LIN {X 0.222,Y -452.244,Z 357.481,A 0.000,B 0.000,C 90.000,E1 266.502} C_DIS
LIN {X -0.089,Y -444.723,Z 357.479,A 0.000,B 0.000,C 90.000,E1 266.274} C_DIS
LIN {X 0.117,Y -436.649,Z 357.478,A 0.000,B 0.000,C 90.000,E1 266.045} C_DIS
LIN {X -0.080,Y -427.748,Z 357.477,A 0.000,B 0.000,C 90.000,E1 265.927} C_DIS
LIN {X 0.197,Y -418.115,Z 357.477,A 0.000,B 0.000,C 90.000,E1 265.812} C_DIS
LIN {X 0.128,Y -415.170,Z 357.477,A 0.000,B 0.000,C 90.000,E1 265.812} C_DIS
LIN {X 0.027,Y -180.914,Z 357.477,A 0.000,B 0.000,C 90.000,E1 265.812} C_DIS
LIN {X -0.032,Y -180.848,Z 357.472,A 0.000,B 0.000,C 90.000,E1 264.951} C_DIS
LIN {X 0.050,Y -178.957,Z 357.444,A 0.000,B 0.000,C 90.000,E1 259.859} C_DIS
LIN {X -0.057,Y -177.360,Z 357.430,A 0.000,B 0.000,C 90.000,E1 257.353} C_DIS
LIN {X 0.039,Y -175.531,Z 357.411,A 0.000,B 0.000,C 90.000,E1 253.921} C_DIS
LIN {X 0.040,Y -172.266,Z 357.387,A 0.000,B 0.000,C 90.000,E1 249.645} C_DIS
LIN {X 0.079,Y -171.746,Z 357.382,A 0.000,B 0.000,C 90.000,E1 248.773} C_DIS
LIN {X -0.063,Y -167.343,Z 357.353,A 0.000,B 0.000,C 90.000,E1 243.640} C_DIS
LIN {X 0.018,Y -166.730,Z 357.349,A 0.000,B 0.000,C 90.000,E1 242.743} C_DIS
LIN {X -0.069,Y -162.709,Z 357.324,A 0.000,B 0.000,C 90.000,E1 238.408} C_DIS
LIN {X -0.007,Y -161.400,Z 357.315,A 0.000,B 0.000,C 90.000,E1 236.628} C_DIS
LIN {X 0.035,Y -157.393,Z 357.290,A 0.000,B 0.000,C 90.000,E1 232.190} C_DIS
LIN {X -0.032,Y -155.390,Z 357.275,A 0.000,B 0.000,C 90.000,E1 229.542} C_DIS
LIN {X 0.007,Y -151.724,Z 357.250,A 0.000,B 0.000,C 90.000,E1 225.040} C_DIS
LIN {X 0.023,Y -149.918,Z 357.235,A 0.000,B 0.000,C 90.000,E1 222.324} C_DIS
LIN {X -0.059,Y -146.773,Z 357.210,A 0.000,B 0.000,C 90.000,E1 217.810} C_DIS
LIN {X 0.045,Y -145.342,Z 357.195,A 0.000,B 0.000,C 90.000,E1 215.025} C_DIS
LIN {X -0.040,Y -142.418,Z 357.164,A 0.000,B 0.000,C 90.000,E1 209.539} C_DIS
LIN {X 0.009,Y -141.404,Z 357.149,A 0.000,B 0.000,C 90.000,E1 206.744} C_DIS
LIN {X -0.003,Y -139.356,Z 357.112,A 0.000,B 0.000,C 90.000,E1 200.248} C_DIS
LIN {X -0.015,Y -138.798,Z 357.097,A 0.000,B 0.000,C 90.000,E1 197.457} C_DIS
LIN {X 0.039,Y -138.348,Z 357.055,A 0.000,B 0.000,C 90.000,E1 189.962} C_DIS
LIN {X 0.057,Y -139.371,Z 357.009,A 0.000,B 0.000,C 90.000,E1 181.547} C_DIS
LIN {X -0.029,Y -141.260,Z 356.973,A 0.000,B 0.000,C 90.000,E1 175.065} C_DIS
LIN {X -0.071,Y -142.628,Z 356.957,A 0.000,B 0.000,C 90.000,E1 172.299} C_DIS
LIN {X 0.022,Y -144.952,Z 356.931,A 0.000,B 0.000,C 90.000,E1 167.645} C_DIS
LIN {X 0.013,Y -147.581,Z 356.911,A 0.000,B 0.000,C 90.000,E1 163.976} C_DIS
LIN {X 0.044,Y -150.192,Z 356.891,A 0.000,B 0.000,C 90.000,E1 160.315} C_DIS
LIN {X -0.030,Y -153.574,Z 356.871,A 0.000,B 0.000,C 90.000,E1 156.719} C_DIS
LIN {X -0.039,Y -156.991,Z 356.851,A 0.000,B 0.000,C 90.000,E1 153.127} C_DIS
LIN {X 0.034,Y -161.105,Z 356.831,A 0.000,B 0.000,C 90.000,E1 149.537} C_DIS
LIN {X -0.021,Y -163.208,Z 356.821,A 0.000,B 0.000,C 90.000,E1 147.788} C_DIS
LIN {X -0.016,Y -167.635,Z 356.802,A 0.000,B 0.000,C 90.000,E1 144.276} C_DIS
LIN {X -0.001,Y -171.461,Z 356.787,A 0.000,B 0.000,C 90.000,E1 141.662} C_DIS
LIN {X -0.071,Y -176.386,Z 356.768,A 0.000,B 0.000,C 90.000,E1 138.243} C_DIS
LIN {X 0.051,Y -180.680,Z 356.754,A 0.000,B 0.000,C 90.000,E1 135.648} C_DIS
LIN {X 0.033,Y -186.082,Z 356.735,A 0.000,B 0.000,C 90.000,E1 132.285} C_DIS
LIN {X -0.030,Y -190.719,Z 356.721,A 0.000,B 0.000,C 90.000,E1 129.806} C_DIS
LIN {X 0.001,Y -196.472,Z 356.703,A 0.000,B 0.000,C 90.000,E1 126.503} C_DIS
LIN {X 0.023,Y -199.896,Z 356.693,A 0.000,B 0.000,C 90.000,E1 124.771} C_DIS
LIN {X -0.019,Y -300.209,Z 356.693,A 0.000,B 0.000,C 90.000,E1 124.771} C_DIS
LIN {X -0.007,Y -301.841,Z 356.693,A 0.000,B 0.000,C 90.000,E1 124.739} C_DIS
LIN {X 0.022,Y -305.622,Z 356.692,A 0.000,B 0.000,C 90.000,E1 124.565} C_DIS
LIN {X -0.029,Y -307.838,Z 356.691,A 0.000,B 0.000,C 90.000,E1 124.405} C_DIS
LIN {X -0.050,Y -310.913,Z 356.689,A 0.000,B 0.000,C 90.000,E1 124.072} C_DIS
LIN {X -0.137,Y -312.908,Z 356.688,A 0.000,B 0.000,C 90.000,E1 123.785} C_DIS
LIN {X 0.036,Y -314.472,Z 356.686,A 0.000,B 0.000,C 90.000,E1 123.452} C_DIS
LIN {X -0.111,Y -316.907,Z 356.682,A 0.000,B 0.000,C 90.000,E1 122.832} C_DIS
LIN {X 0.081,Y -327.434,Z 356.666,A 0.000,B 0.000,C 90.000,E1 119.922} C_DIS
LIN {X -0.084,Y -339.335,Z 356.651,A 0.000,B 0.000,C 90.000,E1 117.129} C_DIS
LIN {X 0.101,Y -352.712,Z 356.635,A 0.000,B 0.000,C 90.000,E1 114.335} C_DIS
LIN {X -0.020,Y -365.944,Z 356.622,A 0.000,B 0.000,C 90.000,E1 111.950} C_DIS
LIN {X 0.123,Y -380.539,Z 356.609,A 0.000,B 0.000,C 90.000,E1 109.577} C_DIS
LIN {X 0.160,Y -396.602,Z 356.596,A 0.000,B 0.000,C 90.000,E1 107.275} C_DIS
LIN {X -0.034,Y -414.254,Z 356.584,A 0.000,B 0.000,C 90.000,E1 105.064} C_DIS
LIN {X 0.018,Y -433.580,Z 356.572,A 0.000,B 0.000,C 90.000,E1 102.883} C_DIS
LIN {X 0.187,Y -453.825,Z 356.560,A 0.000,B 0.000,C 90.000,E1 100.838} C_DIS
LIN {X -0.188,Y -474.606,Z 356.550,A 0.000,B 0.000,C 90.000,E1 99.029} C_DIS
LIN {X -0.195,Y -492.986,Z 356.542,A 0.000,B 0.000,C 90.000,E1 97.530} C_DIS
LIN {X 0.033,Y -496.458,Z 356.539,A 0.000,B 0.000,C 90.000,E1 97.068} C_DIS
LIN {X -0.061,Y -497.755,Z 356.538,A 0.000,B 0.000,C 90.000,E1 96.834} C_DIS
LIN {X -0.215,Y -498.705,Z 356.537,A 0.000,B 0.000,C 90.000,E1 96.606} C_DIS
LIN {X 0.058,Y -499.740,Z 356.534,A 0.000,B 0.000,C 90.000,E1 96.087} C_DIS
LIN {X -0.161,Y -499.759,Z 356.531,A 0.000,B 0.000,C 90.000,E1 95.625} C_DIS
LIN {X 0.121,Y -498.765,Z 356.528,A 0.000,B 0.000,C 90.000,E1 95.106} C_DIS
LIN {X -0.008,Y -497.842,Z 356.527,A 0.000,B 0.000,C 90.000,E1 94.878} C_DIS
LIN {X -0.095,Y -496.578,Z 356.526,A 0.000,B 0.000,C 90.000,E1 94.645} C_DIS
LIN {X 0.031,Y -491.350,Z 356.522,A 0.000,B 0.000,C 90.000,E1 93.898} C_DIS
LIN {X -0.040,Y -483.657,Z 356.516,A 0.000,B 0.000,C 90.000,E1 92.922} C_DIS
LIN {X 0.090,Y -463.710,Z 356.502,A 0.000,B 0.000,C 90.000,E1 90.401} C_DIS
LIN {X 0.125,Y -445.143,Z 356.488,A 0.000,B 0.000,C 90.000,E1 87.822} C_DIS
LIN {X -0.162,Y -426.612,Z 356.472,A 0.000,B 0.000,C 90.000,E1 84.951} C_DIS
LIN {X 0.108,Y -406.776,Z 356.452,A 0.000,B 0.000,C 90.000,E1 81.376} C_DIS
LIN {X -0.002,Y -395.068,Z 356.440,A 0.000,B 0.000,C 90.000,E1 79.162} C_DIS
LIN {X 0.039,Y -384.866,Z 356.429,A 0.000,B 0.000,C 90.000,E1 77.173} C_DIS
LIN {X 0.046,Y -373.237,Z 356.416,A 0.000,B 0.000,C 90.000,E1 74.866} C_DIS
LIN {X -0.124,Y -361.668,Z 356.403,A 0.000,B 0.000,C 90.000,E1 72.543} C_DIS
LIN {X 0.054,Y -351.512,Z 356.391,A 0.000,B 0.000,C 90.000,E1 70.423} C_DIS
LIN {X 0.148,Y -337.364,Z 356.374,A 0.000,B 0.000,C 90.000,E1 67.358} C_DIS
LIN {X -0.164,Y -326.775,Z 356.361,A 0.000,B 0.000,C 90.000,E1 64.921} C_DIS
LIN {X 0.063,Y -315.883,Z 356.345,A 0.000,B 0.000,C 90.000,E1 62.025} C_DIS
LIN {X 0.088,Y -303.361,Z 356.325,A 0.000,B 0.000,C 90.000,E1 58.456} C_DIS
LIN {X -0.062,Y -291.846,Z 356.305,A 0.000,B 0.000,C 90.000,E1 54.848} C_DIS
LIN {X 0.046,Y -282.258,Z 356.286,A 0.000,B 0.000,C 90.000,E1 51.457} C_DIS
LIN {X -0.006,Y -274.758,Z 356.271,A 0.000,B 0.000,C 90.000,E1 48.728} C_DIS
LIN {X -0.073,Y -269.054,Z 356.259,A 0.000,B 0.000,C 90.000,E1 46.662} C_DIS
LIN {X -0.126,Y -261.490,Z 356.244,A 0.000,B 0.000,C 90.000,E1 43.866} C_DIS
LIN {X 0.125,Y -255.793,Z 356.232,A 0.000,B 0.000,C 90.000,E1 41.676} C_DIS
LIN {X -0.072,Y -250.024,Z 356.220,A 0.000,B 0.000,C 90.000,E1 39.564} C_DIS
LIN {X 0.010,Y -244.096,Z 356.208,A 0.000,B 0.000,C 90.000,E1 37.363} C_DIS
LIN {X 0.041,Y -236.316,Z 356.191,A 0.000,B 0.000,C 90.000,E1 34.405} C_DIS
LIN {X 0.010,Y -228.739,Z 356.175,A 0.000,B 0.000,C 90.000,E1 31.416} C_DIS
LIN {X 0.063,Y -221.644,Z 356.158,A 0.000,B 0.000,C 90.000,E1 28.359} C_DIS
LIN {X -0.026,Y -213.645,Z 356.136,A 0.000,B 0.000,C 90.000,E1 24.515} C_DIS
LIN {X 0.048,Y -207.922,Z 356.119,A 0.000,B 0.000,C 90.000,E1 21.354} C_DIS
LIN {X 0.025,Y -202.976,Z 356.101,A 0.000,B 0.000,C 90.000,E1 18.181} C_DIS
LIN {X 0.076,Y -198.614,Z 356.083,A 0.000,B 0.000,C 90.000,E1 14.954} C_DIS
LIN {X 0.078,Y -194.085,Z 356.061,A 0.000,B 0.000,C 90.000,E1 10.894} C_DIS
LIN {X -0.046,Y -190.735,Z 356.038,A 0.000,B 0.000,C 90.000,E1 6.834} C_DIS
LIN {X 0.022,Y -188.091,Z 356.006,A 0.000,B 0.000,C 90.000,E1 1.031} C_DIS
LIN {X 0.029,Y -189.258,Z 355.942,A 0.000,B 0.000,C 90.000,E1 349.567} C_DIS
LIN {X -0.030,Y -192.110,Z 355.915,A 0.000,B 0.000,C 90.000,E1 344.629} C_DIS
LIN {X 0.073,Y -195.713,Z 355.892,A 0.000,B 0.000,C 90.000,E1 340.496} C_DIS
LIN {X 0.058,Y -200.400,Z 355.869,A 0.000,B 0.000,C 90.000,E1 336.433} C_DIS
LIN {X 0.058,Y -206.128,Z 355.847,A 0.000,B 0.000,C 90.000,E1 332.410} C_DIS
LIN {X -0.011,Y -212.845,Z 355.825,A 0.000,B 0.000,C 90.000,E1 328.456} C_DIS
LIN {X -0.091,Y -220.250,Z 355.803,A 0.000,B 0.000,C 90.000,E1 324.562} C_DIS
LIN {X 0.033,Y -228.477,Z 355.782,A 0.000,B 0.000,C 90.000,E1 320.678} C_DIS
LIN {X 0.079,Y -235.880,Z 355.765,A 0.000,B 0.000,C 90.000,E1 317.634} C_DIS
LIN {X 0.126,Y -245.235,Z 355.746,A 0.000,B 0.000,C 90.000,E1 314.271} C_DIS
LIN {X 0.123,Y -255.868,Z 355.728,A 0.000,B 0.000,C 90.000,E1 310.987} C_DIS
LIN {X -0.051,Y -267.304,Z 355.710,A 0.000,B 0.000,C 90.000,E1 307.810} C_DIS
LIN {X -0.024,Y -279.759,Z 355.693,A 0.000,B 0.000,C 90.000,E1 304.659} C_DIS
LIN {X -0.037,Y -293.589,Z 355.675,A 0.000,B 0.000,C 90.000,E1 301.592} C_DIS
LIN {X -0.071,Y -310.841,Z 355.657,A 0.000,B 0.000,C 90.000,E1 298.281} C_DIS
LIN {X -0.109,Y -320.424,Z 355.648,A 0.000,B 0.000,C 90.000,E1 296.668} C_DIS
LIN {X -0.141,Y -341.506,Z 355.630,A 0.000,B 0.000,C 90.000,E1 293.515} C_DIS
LIN {X -0.076,Y -354.944,Z 355.620,A 0.000,B 0.000,C 90.000,E1 291.663} C_DIS
LIN {X -0.135,Y -371.202,Z 355.609,A 0.000,B 0.000,C 90.000,E1 289.577} C_DIS
LIN {X -0.110,Y -393.867,Z 355.594,A 0.000,B 0.000,C 90.000,E1 286.968} C_DIS
LIN {X 0.192,Y -411.753,Z 355.584,A 0.000,B 0.000,C 90.000,E1 285.009} C_DIS
LIN {X 0.049,Y -424.400,Z 355.576,A 0.000,B 0.000,C 90.000,E1 283.703} C_DIS
LIN {X -0.042,Y -434.234,Z 355.570,A 0.000,B 0.000,C 90.000,E1 282.647} C_DIS
LIN {X 0.113,Y -441.110,Z 355.566,A 0.000,B 0.000,C 90.000,E1 281.827} C_DIS
LIN {X -0.197,Y -447.486,Z 355.561,A 0.000,B 0.000,C 90.000,E1 281.074} C_DIS
LIN {X -0.116,Y -455.315,Z 355.556,A 0.000,B 0.000,C 90.000,E1 280.018} C_DIS
LIN {X -0.024,Y -462.550,Z 355.550,A 0.000,B 0.000,C 90.000,E1 278.973} C_DIS
LIN {X 0.089,Y -469.119,Z 355.544,A 0.000,B 0.000,C 90.000,E1 277.936} C_DIS
LIN {X -0.125,Y -475.245,Z 355.539,A 0.000,B 0.000,C 90.000,E1 276.947} C_DIS
LIN {X -0.194,Y -479.378,Z 355.534,A 0.000,B 0.000,C 90.000,E1 276.201} C_DIS
LIN {X -0.180,Y -482.963,Z 355.530,A 0.000,B 0.000,C 90.000,E1 275.448} C_DIS
LIN {X -0.051,Y -484.974,Z 355.527,A 0.000,B 0.000,C 90.000,E1 274.935} C_DIS
LIN {X 0.129,Y -486.567,Z 355.525,A 0.000,B 0.000,C 90.000,E1 274.416} C_DIS
LIN {X -0.167,Y -487.736,Z 355.522,A 0.000,B 0.000,C 90.000,E1 273.955} C_DIS
LIN {X -0.001,Y -488.552,Z 355.519,A 0.000,B 0.000,C 90.000,E1 273.440} C_DIS
LIN {X 0.202,Y -489.054,Z 355.516,A 0.000,B 0.000,C 90.000,E1 272.922} C_DIS
LIN {X -0.104,Y -489.200,Z 355.514,A 0.000,B 0.000,C 90.000,E1 272.465} C_DIS
LIN {X 0.084,Y -489.089,Z 355.511,A 0.000,B 0.000,C 90.000,E1 271.949} C_DIS
LIN {X -0.201,Y -488.696,Z 355.508,A 0.000,B 0.000,C 90.000,E1 271.489} C_DIS
LIN {X -0.012,Y -487.974,Z 355.505,A 0.000,B 0.000,C 90.000,E1 270.974} C_DIS
LIN {X 0.174,Y -486.933,Z 355.503,A 0.000,B 0.000,C 90.000,E1 270.458} C_DIS
LIN {X -0.129,Y -485.506,Z 355.500,A 0.000,B 0.000,C 90.000,E1 270.000} C_DIS
LIN {X 0.048,Y -483.635,Z 355.497,A 0.000,B 0.000,C 90.000,E1 269.484} C_DIS
LIN {X 0.214,Y -481.141,Z 355.494,A 0.000,B 0.000,C 90.000,E1 268.969} C_DIS
LIN {X -0.118,Y -477.917,Z 355.492,A 0.000,B 0.000,C 90.000,E1 268.511} C_DIS
LIN {X 0.027,Y -473.725,Z 355.489,A 0.000,B 0.000,C 90.000,E1 267.993} C_DIS
LIN {X -0.155,Y -471.235,Z 355.487,A 0.000,B 0.000,C 90.000,E1 267.764} C_DIS
LIN {X 0.146,Y -465.489,Z 355.485,A 0.000,B 0.000,C 90.000,E1 267.249} C_DIS
LIN {X 0.159,Y -462.172,Z 355.484,A 0.000,B 0.000,C 90.000,E1 267.020} C_DIS
LIN {X -0.137,Y -455.260,Z 355.481,A 0.000,B 0.000,C 90.000,E1 266.674} C_DIS
LIN {X 0.143,Y -447.669,Z 355.480,A 0.000,B 0.000,C 90.000,E1 266.331} C_DIS
LIN {X 0.101,Y -439.662,Z 355.478,A 0.000,B 0.000,C 90.000,E1 266.102} C_DIS
LIN {X 0.154,Y -430.752,Z 355.477,A 0.000,B 0.000,C 90.000,E1 265.927} C_DIS
LIN {X 0.176,Y -420.110,Z 355.477,A 0.000,B 0.000,C 90.000,E1 265.812} C_DIS
LIN {X 0.111,Y -417.514,Z 355.477,A 0.000,B 0.000,C 90.000,E1 265.812} C_DIS
LIN {X 0.020,Y -180.914,Z 355.477,A 0.000,B 0.000,C 90.000,E1 265.812} C_DIS
LIN {X -0.087,Y -180.842,Z 355.472,A 0.000,B 0.000,C 90.000,E1 264.951} C_DIS
LIN {X -0.005,Y -178.951,Z 355.444,A 0.000,B 0.000,C 90.000,E1 259.859} C_DIS
LIN {X 0.012,Y -176.857,Z 355.425,A 0.000,B 0.000,C 90.000,E1 256.464} C_DIS
LIN {X -0.015,Y -175.518,Z 355.411,A 0.000,B 0.000,C 90.000,E1 253.921} C_DIS
LIN {X -0.013,Y -172.255,Z 355.387,A 0.000,B 0.000,C 90.000,E1 249.645} C_DIS
LIN {X 0.025,Y -171.734,Z 355.382,A 0.000,B 0.000,C 90.000,E1 248.773} C_DIS
LIN {X 0.033,Y -167.331,Z 355.353,A 0.000,B 0.000,C 90.000,E1 243.589} C_DIS
LIN {X -0.034,Y -166.715,Z 355.349,A 0.000,B 0.000,C 90.000,E1 242.743} C_DIS
LIN {X 0.104,Y -162.695,Z 355.324,A 0.000,B 0.000,C 90.000,E1 238.329} C_DIS
LIN {X -0.059,Y -161.385,Z 355.314,A 0.000,B 0.000,C 90.000,E1 236.628} C_DIS
LIN {X -0.016,Y -157.379,Z 355.290,A 0.000,B 0.000,C 90.000,E1 232.190} C_DIS
LIN {X -0.082,Y -155.372,Z 355.275,A 0.000,B 0.000,C 90.000,E1 229.542} C_DIS
LIN {X 0.065,Y -151.711,Z 355.250,A 0.000,B 0.000,C 90.000,E1 225.000} C_DIS
LIN {X -0.027,Y -149.903,Z 355.235,A 0.000,B 0.000,C 90.000,E1 222.324} C_DIS
LIN {X 0.009,Y -146.762,Z 355.210,A 0.000,B 0.000,C 90.000,E1 217.764} C_DIS
LIN {X -0.003,Y -145.329,Z 355.195,A 0.000,B 0.000,C 90.000,E1 215.025} C_DIS
LIN {X 0.036,Y -142.411,Z 355.164,A 0.000,B 0.000,C 90.000,E1 209.489} C_DIS
LIN {X -0.037,Y -141.395,Z 355.148,A 0.000,B 0.000,C 90.000,E1 206.744} C_DIS
LIN {X -0.050,Y -139.354,Z 355.112,A 0.000,B 0.000,C 90.000,E1 200.248} C_DIS
LIN {X -0.062,Y -138.794,Z 355.097,A 0.000,B 0.000,C 90.000,E1 197.457} C_DIS
LIN {X -0.007,Y -138.346,Z 355.055,A 0.000,B 0.000,C 90.000,E1 189.962} C_DIS
LIN {X 0.010,Y -139.378,Z 355.009,A 0.000,B 0.000,C 90.000,E1 181.547} C_DIS
LIN {X 0.064,Y -141.269,Z 354.972,A 0.000,B 0.000,C 90.000,E1 175.008} C_DIS
LIN {X 0.022,Y -142.635,Z 354.957,A 0.000,B 0.000,C 90.000,E1 172.243} C_DIS
LIN {X -0.026,Y -144.964,Z 354.931,A 0.000,B 0.000,C 90.000,E1 167.645} C_DIS
LIN {X -0.036,Y -147.592,Z 354.911,A 0.000,B 0.000,C 90.000,E1 163.976} C_DIS
LIN {X -0.006,Y -150.208,Z 354.891,A 0.000,B 0.000,C 90.000,E1 160.315} C_DIS
LIN {X 0.061,Y -153.593,Z 354.870,A 0.000,B 0.000,C 90.000,E1 156.666} C_DIS
LIN {X 0.050,Y -157.010,Z 354.851,A 0.000,B 0.000,C 90.000,E1 153.076} C_DIS
LIN {X -0.017,Y -161.128,Z 354.831,A 0.000,B 0.000,C 90.000,E1 149.537} C_DIS
LIN {X -0.073,Y -163.228,Z 354.821,A 0.000,B 0.000,C 90.000,E1 147.788} C_DIS
LIN {X -0.069,Y -167.661,Z 354.801,A 0.000,B 0.000,C 90.000,E1 144.276} C_DIS
LIN {X 0.080,Y -171.484,Z 354.787,A 0.000,B 0.000,C 90.000,E1 141.618} C_DIS
LIN {X 0.124,Y -176.414,Z 354.768,A 0.000,B 0.000,C 90.000,E1 138.162} C_DIS
LIN {X -0.005,Y -180.709,Z 354.754,A 0.000,B 0.000,C 90.000,E1 135.648} C_DIS
LIN {X -0.023,Y -186.112,Z 354.735,A 0.000,B 0.000,C 90.000,E1 132.285} C_DIS
LIN {X 0.035,Y -190.750,Z 354.721,A 0.000,B 0.000,C 90.000,E1 129.769} C_DIS
LIN {X -0.056,Y -196.504,Z 354.703,A 0.000,B 0.000,C 90.000,E1 126.503} C_DIS
LIN {X -0.028,Y -199.994,Z 354.693,A 0.000,B 0.000,C 90.000,E1 124.739} C_DIS
LIN {X -0.095,Y -300.284,Z 354.693,A 0.000,B 0.000,C 90.000,E1 124.739} C_DIS
LIN {X 0.105,Y -305.259,Z 354.692,A 0.000,B 0.000,C 90.000,E1 124.532} C_DIS
LIN {X -0.119,Y -307.624,Z 354.691,A 0.000,B 0.000,C 90.000,E1 124.405} C_DIS
LIN {X 0.033,Y -310.819,Z 354.689,A 0.000,B 0.000,C 90.000,E1 124.040} C_DIS
LIN {X -0.183,Y -312.817,Z 354.688,A 0.000,B 0.000,C 90.000,E1 123.785} C_DIS
LIN {X 0.038,Y -314.388,Z 354.686,A 0.000,B 0.000,C 90.000,E1 123.452} C_DIS
LIN {X -0.168,Y -315.763,Z 354.684,A 0.000,B 0.000,C 90.000,E1 123.166} C_DIS
LIN {X 0.081,Y -327.412,Z 354.666,A 0.000,B 0.000,C 90.000,E1 119.922} C_DIS
LIN {X -0.084,Y -339.313,Z 354.651,A 0.000,B 0.000,C 90.000,E1 117.129} C_DIS
LIN {X 0.100,Y -352.690,Z 354.635,A 0.000,B 0.000,C 90.000,E1 114.335} C_DIS
LIN {X -0.022,Y -365.922,Z 354.622,A 0.000,B 0.000,C 90.000,E1 111.950} C_DIS
LIN {X 0.121,Y -380.516,Z 354.609,A 0.000,B 0.000,C 90.000,E1 109.577} C_DIS
LIN {X 0.157,Y -396.579,Z 354.596,A 0.000,B 0.000,C 90.000,E1 107.275} C_DIS
LIN {X -0.039,Y -414.231,Z 354.584,A 0.000,B 0.000,C 90.000,E1 105.064} C_DIS
LIN {X 0.013,Y -433.557,Z 354.572,A 0.000,B 0.000,C 90.000,E1 102.883} C_DIS
LIN {X 0.182,Y -453.803,Z 354.560,A 0.000,B 0.000,C 90.000,E1 100.838} C_DIS
LIN {X -0.193,Y -474.583,Z 354.550,A 0.000,B 0.000,C 90.000,E1 99.029} C_DIS
LIN {X -0.202,Y -493.003,Z 354.542,A 0.000,B 0.000,C 90.000,E1 97.530} C_DIS
LIN {X 0.066,Y -496.517,Z 354.539,A 0.000,B 0.000,C 90.000,E1 97.068} C_DIS
LIN {X -0.028,Y -497.848,Z 354.538,A 0.000,B 0.000,C 90.000,E1 96.834} C_DIS
LIN {X -0.183,Y -498.825,Z 354.537,A 0.000,B 0.000,C 90.000,E1 96.606} C_DIS
LIN {X 0.091,Y -499.906,Z 354.534,A 0.000,B 0.000,C 90.000,E1 96.087} C_DIS
LIN {X -0.127,Y -499.966,Z 354.531,A 0.000,B 0.000,C 90.000,E1 95.625} C_DIS
LIN {X 0.157,Y -499.015,Z 354.528,A 0.000,B 0.000,C 90.000,E1 95.106} C_DIS
LIN {X -0.058,Y -496.885,Z 354.526,A 0.000,B 0.000,C 90.000,E1 94.645} C_DIS
LIN {X 0.075,Y -491.707,Z 354.522,A 0.000,B 0.000,C 90.000,E1 93.898} C_DIS
LIN {X 0.007,Y -484.011,Z 354.516,A 0.000,B 0.000,C 90.000,E1 92.922} C_DIS
LIN {X -0.119,Y -465.981,Z 354.504,A 0.000,B 0.000,C 90.000,E1 90.688} C_DIS
LIN {X 0.187,Y -445.441,Z 354.488,A 0.000,B 0.000,C 90.000,E1 87.822} C_DIS
LIN {X -0.095,Y -426.896,Z 354.472,A 0.000,B 0.000,C 90.000,E1 84.951} C_DIS
LIN {X 0.133,Y -408.516,Z 354.454,A 0.000,B 0.000,C 90.000,E1 81.659} C_DIS
LIN {X 0.002,Y -396.827,Z 354.441,A 0.000,B 0.000,C 90.000,E1 79.454} C_DIS
LIN {X 0.074,Y -386.615,Z 354.430,A 0.000,B 0.000,C 90.000,E1 77.465} C_DIS
LIN {X 0.029,Y -374.970,Z 354.418,A 0.000,B 0.000,C 90.000,E1 75.172} C_DIS
LIN {X 0.000,Y -363.392,Z 354.405,A 0.000,B 0.000,C 90.000,E1 72.834} C_DIS
LIN {X 0.106,Y -353.238,Z 354.393,A 0.000,B 0.000,C 90.000,E1 70.732} C_DIS
LIN {X -0.076,Y -340.347,Z 354.378,A 0.000,B 0.000,C 90.000,E1 68.028} C_DIS
LIN {X -0.062,Y -327.003,Z 354.361,A 0.000,B 0.000,C 90.000,E1 64.921} C_DIS
LIN {X 0.169,Y -316.120,Z 354.345,A 0.000,B 0.000,C 90.000,E1 62.025} C_DIS
LIN {X 0.037,Y -303.593,Z 354.325,A 0.000,B 0.000,C 90.000,E1 58.486} C_DIS
LIN {X 0.049,Y -292.083,Z 354.305,A 0.000,B 0.000,C 90.000,E1 54.848} C_DIS
LIN {X 0.162,Y -282.468,Z 354.286,A 0.000,B 0.000,C 90.000,E1 51.457} C_DIS
LIN {X -0.095,Y -274.971,Z 354.271,A 0.000,B 0.000,C 90.000,E1 48.771} C_DIS
LIN {X 0.047,Y -269.274,Z 354.259,A 0.000,B 0.000,C 90.000,E1 46.662} C_DIS
LIN {X -0.005,Y -261.712,Z 354.244,A 0.000,B 0.000,C 90.000,E1 43.866} C_DIS
LIN {X -0.113,Y -256.022,Z 354.232,A 0.000,B 0.000,C 90.000,E1 41.757} C_DIS
LIN {X 0.052,Y -250.276,Z 354.220,A 0.000,B 0.000,C 90.000,E1 39.564} C_DIS
LIN {X -0.012,Y -244.346,Z 354.208,A 0.000,B 0.000,C 90.000,E1 37.397} C_DIS
LIN {X -0.027,Y -236.544,Z 354.191,A 0.000,B 0.000,C 90.000,E1 34.452} C_DIS
LIN {X -0.056,Y -228.952,Z 354.175,A 0.000,B 0.000,C 90.000,E1 31.465} C_DIS
LIN {X -0.002,Y -221.843,Z 354.158,A 0.000,B 0.000,C 90.000,E1 28.409} C_DIS
LIN {X -0.052,Y -215.344,Z 354.141,A 0.000,B 0.000,C 90.000,E1 25.335} C_DIS
LIN {X -0.049,Y -209.426,Z 354.123,A 0.000,B 0.000,C 90.000,E1 22.206} C_DIS
LIN {X -0.035,Y -204.266,Z 354.106,A 0.000,B 0.000,C 90.000,E1 19.033} C_DIS
LIN {X 0.015,Y -198.736,Z 354.083,A 0.000,B 0.000,C 90.000,E1 15.009} C_DIS
LIN {X 0.020,Y -194.182,Z 354.061,A 0.000,B 0.000,C 90.000,E1 10.950} C_DIS
LIN {X 0.086,Y -190.816,Z 354.038,A 0.000,B 0.000,C 90.000,E1 6.834} C_DIS
LIN {X -0.032,Y -188.135,Z 354.006,A 0.000,B 0.000,C 90.000,E1 1.088} C_DIS
LIN {X 0.032,Y -189.256,Z 353.942,A 0.000,B 0.000,C 90.000,E1 349.567} C_DIS
LIN {X -0.027,Y -192.100,Z 353.915,A 0.000,B 0.000,C 90.000,E1 344.629} C_DIS
LIN {X 0.075,Y -195.701,Z 353.892,A 0.000,B 0.000,C 90.000,E1 340.496} C_DIS
LIN {X 0.061,Y -200.354,Z 353.869,A 0.000,B 0.000,C 90.000,E1 336.433} C_DIS
LIN {X 0.058,Y -206.079,Z 353.847,A 0.000,B 0.000,C 90.000,E1 332.410} C_DIS
LIN {X -0.013,Y -212.754,Z 353.825,A 0.000,B 0.000,C 90.000,E1 328.456} C_DIS
LIN {X 0.029,Y -218.624,Z 353.807,A 0.000,B 0.000,C 90.000,E1 325.308} C_DIS
LIN {X -0.024,Y -226.678,Z 353.786,A 0.000,B 0.000,C 90.000,E1 321.457} C_DIS
LIN {X 0.003,Y -233.882,Z 353.769,A 0.000,B 0.000,C 90.000,E1 318.405} C_DIS
LIN {X -0.015,Y -243.005,Z 353.750,A 0.000,B 0.000,C 90.000,E1 315.040} C_DIS
LIN {X -0.096,Y -253.346,Z 353.732,A 0.000,B 0.000,C 90.000,E1 311.757} C_DIS
LIN {X 0.136,Y -263.322,Z 353.716,A 0.000,B 0.000,C 90.000,E1 308.830} C_DIS
LIN {X 0.065,Y -275.457,Z 353.698,A 0.000,B 0.000,C 90.000,E1 305.678} C_DIS
LIN {X -0.147,Y -288.849,Z 353.681,A 0.000,B 0.000,C 90.000,E1 302.625} C_DIS
LIN {X -0.062,Y -302.152,Z 353.666,A 0.000,B 0.000,C 90.000,E1 299.922} C_DIS
LIN {X -0.145,Y -314.744,Z 353.653,A 0.000,B 0.000,C 90.000,E1 297.641} C_DIS
LIN {X 0.156,Y -330.965,Z 353.639,A 0.000,B 0.000,C 90.000,E1 295.027} C_DIS
LIN {X -0.130,Y -350.726,Z 353.624,A 0.000,B 0.000,C 90.000,E1 292.280} C_DIS
LIN {X -0.130,Y -371.488,Z 353.609,A 0.000,B 0.000,C 90.000,E1 289.577} C_DIS
LIN {X 0.143,Y -391.527,Z 353.596,A 0.000,B 0.000,C 90.000,E1 287.221} C_DIS
LIN {X 0.076,Y -409.419,Z 353.585,A 0.000,B 0.000,C 90.000,E1 285.300} C_DIS
LIN {X -0.129,Y -421.983,Z 353.578,A 0.000,B 0.000,C 90.000,E1 284.008} C_DIS
LIN {X -0.165,Y -431.880,Z 353.572,A 0.000,B 0.000,C 90.000,E1 282.939} C_DIS
LIN {X -0.042,Y -438.931,Z 353.567,A 0.000,B 0.000,C 90.000,E1 282.119} C_DIS
LIN {X 0.156,Y -445.458,Z 353.563,A 0.000,B 0.000,C 90.000,E1 281.299} C_DIS
LIN {X 0.134,Y -453.365,Z 353.557,A 0.000,B 0.000,C 90.000,E1 280.254} C_DIS
LIN {X 0.208,Y -460.718,Z 353.551,A 0.000,B 0.000,C 90.000,E1 279.208} C_DIS
LIN {X -0.091,Y -467.436,Z 353.546,A 0.000,B 0.000,C 90.000,E1 278.219} C_DIS
LIN {X 0.081,Y -473.660,Z 353.540,A 0.000,B 0.000,C 90.000,E1 277.182} C_DIS
LIN {X 0.051,Y -477.934,Z 353.536,A 0.000,B 0.000,C 90.000,E1 276.429} C_DIS
LIN {X 0.009,Y -481.718,Z 353.532,A 0.000,B 0.000,C 90.000,E1 275.682} C_DIS
LIN {X -0.001,Y -484.857,Z 353.527,A 0.000,B 0.000,C 90.000,E1 274.935} C_DIS
LIN {X 0.179,Y -486.419,Z 353.525,A 0.000,B 0.000,C 90.000,E1 274.416} C_DIS
LIN {X -0.118,Y -487.618,Z 353.522,A 0.000,B 0.000,C 90.000,E1 273.955} C_DIS
LIN {X 0.047,Y -488.432,Z 353.519,A 0.000,B 0.000,C 90.000,E1 273.440} C_DIS
LIN {X 0.250,Y -488.888,Z 353.516,A 0.000,B 0.000,C 90.000,E1 272.922} C_DIS
LIN {X -0.057,Y -489.031,Z 353.514,A 0.000,B 0.000,C 90.000,E1 272.465} C_DIS
LIN {X 0.130,Y -488.908,Z 353.511,A 0.000,B 0.000,C 90.000,E1 271.949} C_DIS
LIN {X -0.155,Y -488.488,Z 353.508,A 0.000,B 0.000,C 90.000,E1 271.489} C_DIS
LIN {X 0.032,Y -487.783,Z 353.505,A 0.000,B 0.000,C 90.000,E1 270.974} C_DIS
LIN {X 0.217,Y -486.766,Z 353.503,A 0.000,B 0.000,C 90.000,E1 270.458} C_DIS
LIN {X -0.087,Y -485.357,Z 353.500,A 0.000,B 0.000,C 90.000,E1 270.000} C_DIS
LIN {X 0.088,Y -483.453,Z 353.497,A 0.000,B 0.000,C 90.000,E1 269.484} C_DIS
LIN {X -0.227,Y -480.993,Z 353.494,A 0.000,B 0.000,C 90.000,E1 269.026} C_DIS
LIN {X -0.079,Y -477.768,Z 353.492,A 0.000,B 0.000,C 90.000,E1 268.511} C_DIS
LIN {X 0.064,Y -473.683,Z 353.489,A 0.000,B 0.000,C 90.000,E1 267.993} C_DIS
LIN {X 0.171,Y -468.368,Z 353.486,A 0.000,B 0.000,C 90.000,E1 267.478} C_DIS
LIN {X 0.153,Y -465.471,Z 353.485,A 0.000,B 0.000,C 90.000,E1 267.249} C_DIS
LIN {X -0.007,Y -458.987,Z 353.482,A 0.000,B 0.000,C 90.000,E1 266.846} C_DIS
LIN {X -0.035,Y -451.885,Z 353.481,A 0.000,B 0.000,C 90.000,E1 266.502} C_DIS
LIN {X 0.090,Y -444.138,Z 353.479,A 0.000,B 0.000,C 90.000,E1 266.216} C_DIS
LIN {X -0.140,Y -435.960,Z 353.478,A 0.000,B 0.000,C 90.000,E1 266.045} C_DIS
LIN {X 0.098,Y -426.898,Z 353.477,A 0.000,B 0.000,C 90.000,E1 265.869} C_DIS
LIN {X 0.092,Y -419.826,Z 353.477,A 0.000,B 0.000,C 90.000,E1 265.812} C_DIS
LIN {X 0.033,Y -417.348,Z 353.477,A 0.000,B 0.000,C 90.000,E1 265.812} C_DIS
LIN {X -0.011,Y -180.913,Z 353.477,A 0.000,B 0.000,C 90.000,E1 265.812} C_DIS
LIN {X 0.078,Y -180.842,Z 353.472,A 0.000,B 0.000,C 90.000,E1 264.894} C_DIS
LIN {X -0.019,Y -178.949,Z 353.444,A 0.000,B 0.000,C 90.000,E1 259.859} C_DIS
LIN {X -0.003,Y -176.854,Z 353.425,A 0.000,B 0.000,C 90.000,E1 256.464} C_DIS
LIN {X -0.031,Y -175.514,Z 353.411,A 0.000,B 0.000,C 90.000,E1 253.921} C_DIS
LIN {X 0.031,Y -172.252,Z 353.387,A 0.000,B 0.000,C 90.000,E1 249.625} C_DIS
LIN {X 0.010,Y -171.730,Z 353.382,A 0.000,B 0.000,C 90.000,E1 248.773} C_DIS
LIN {X 0.019,Y -167.327,Z 353.353,A 0.000,B 0.000,C 90.000,E1 243.589} C_DIS
LIN {X -0.049,Y -166.711,Z 353.348,A 0.000,B 0.000,C 90.000,E1 242.743} C_DIS
LIN {X 0.089,Y -162.691,Z 353.324,A 0.000,B 0.000,C 90.000,E1 238.329} C_DIS
LIN {X -0.073,Y -161.382,Z 353.314,A 0.000,B 0.000,C 90.000,E1 236.628} C_DIS
LIN {X -0.030,Y -157.375,Z 353.290,A 0.000,B 0.000,C 90.000,E1 232.190} C_DIS
LIN {X 0.004,Y -155.368,Z 353.275,A 0.000,B 0.000,C 90.000,E1 229.504} C_DIS
LIN {X 0.052,Y -151.708,Z 353.250,A 0.000,B 0.000,C 90.000,E1 225.000} C_DIS
LIN {X 0.061,Y -149.899,Z 353.235,A 0.000,B 0.000,C 90.000,E1 222.285} C_DIS
LIN {X 0.085,Y -146.758,Z 353.210,A 0.000,B 0.000,C 90.000,E1 217.729} C_DIS
LIN {X -0.017,Y -145.325,Z 353.195,A 0.000,B 0.000,C 90.000,E1 215.025} C_DIS
LIN {X 0.023,Y -142.409,Z 353.164,A 0.000,B 0.000,C 90.000,E1 209.489} C_DIS
LIN {X -0.051,Y -141.393,Z 353.148,A 0.000,B 0.000,C 90.000,E1 206.744} C_DIS
LIN {X -0.063,Y -139.352,Z 353.112,A 0.000,B 0.000,C 90.000,E1 200.248} C_DIS
LIN {X 0.058,Y -138.792,Z 353.097,A 0.000,B 0.000,C 90.000,E1 197.402} C_DIS
LIN {X -0.020,Y -138.346,Z 353.055,A 0.000,B 0.000,C 90.000,E1 189.962} C_DIS
LIN {X -0.003,Y -139.380,Z 353.009,A 0.000,B 0.000,C 90.000,E1 181.547} C_DIS
LIN {X 0.050,Y -141.271,Z 352.972,A 0.000,B 0.000,C 90.000,E1 175.008} C_DIS
LIN {X 0.009,Y -142.637,Z 352.957,A 0.000,B 0.000,C 90.000,E1 172.243} C_DIS
LIN {X -0.040,Y -144.967,Z 352.931,A 0.000,B 0.000,C 90.000,E1 167.645} C_DIS
LIN {X -0.049,Y -147.595,Z 352.911,A 0.000,B 0.000,C 90.000,E1 163.976} C_DIS
LIN {X -0.020,Y -150.212,Z 352.891,A 0.000,B 0.000,C 90.000,E1 160.315} C_DIS
LIN {X 0.047,Y -153.599,Z 352.870,A 0.000,B 0.000,C 90.000,E1 156.666} C_DIS
LIN {X 0.035,Y -157.015,Z 352.850,A 0.000,B 0.000,C 90.000,E1 153.076} C_DIS
LIN {X -0.032,Y -161.134,Z 352.831,A 0.000,B 0.000,C 90.000,E1 149.537} C_DIS
LIN {X 0.051,Y -163.234,Z 352.821,A 0.000,B 0.000,C 90.000,E1 147.740} C_DIS
LIN {X -0.083,Y -167.667,Z 352.801,A 0.000,B 0.000,C 90.000,E1 144.276} C_DIS
LIN {X 0.064,Y -171.490,Z 352.787,A 0.000,B 0.000,C 90.000,E1 141.618} C_DIS
LIN {X 0.108,Y -176.422,Z 352.768,A 0.000,B 0.000,C 90.000,E1 138.162} C_DIS
LIN {X -0.020,Y -180.717,Z 352.754,A 0.000,B 0.000,C 90.000,E1 135.648} C_DIS
LIN {X -0.039,Y -186.120,Z 352.735,A 0.000,B 0.000,C 90.000,E1 132.285} C_DIS
LIN {X 0.018,Y -190.758,Z 352.721,A 0.000,B 0.000,C 90.000,E1 129.769} C_DIS
LIN {X -0.073,Y -196.513,Z 352.703,A 0.000,B 0.000,C 90.000,E1 126.503} C_DIS
LIN {X -0.010,Y -200.082,Z 352.693,A 0.000,B 0.000,C 90.000,E1 124.692} C_DIS
LIN {X -0.066,Y -299.742,Z 352.693,A 0.000,B 0.000,C 90.000,E1 124.692} C_DIS
LIN {X -0.049,Y -301.869,Z 352.693,A 0.000,B 0.000,C 90.000,E1 124.659} C_DIS
LIN {X 0.106,Y -307.662,Z 352.691,A 0.000,B 0.000,C 90.000,E1 124.326} C_DIS
LIN {X 0.007,Y -310.629,Z 352.689,A 0.000,B 0.000,C 90.000,E1 124.040} C_DIS
LIN {X -0.173,Y -312.662,Z 352.688,A 0.000,B 0.000,C 90.000,E1 123.785} C_DIS
LIN {X 0.082,Y -314.261,Z 352.686,A 0.000,B 0.000,C 90.000,E1 123.452} C_DIS
LIN {X -0.125,Y -315.691,Z 352.684,A 0.000,B 0.000,C 90.000,E1 123.166} C_DIS
LIN {X 0.123,Y -327.361,Z 352.666,A 0.000,B 0.000,C 90.000,E1 119.922} C_DIS
LIN {X -0.041,Y -339.258,Z 352.651,A 0.000,B 0.000,C 90.000,E1 117.129} C_DIS
LIN {X 0.144,Y -352.630,Z 352.635,A 0.000,B 0.000,C 90.000,E1 114.335} C_DIS
LIN {X -0.115,Y -365.858,Z 352.622,A 0.000,B 0.000,C 90.000,E1 111.972} C_DIS
LIN {X 0.164,Y -380.447,Z 352.609,A 0.000,B 0.000,C 90.000,E1 109.577} C_DIS
LIN {X 0.200,Y -396.507,Z 352.596,A 0.000,B 0.000,C 90.000,E1 107.275} C_DIS
LIN {X 0.005,Y -414.154,Z 352.584,A 0.000,B 0.000,C 90.000,E1 105.064} C_DIS
LIN {X 0.057,Y -433.475,Z 352.572,A 0.000,B 0.000,C 90.000,E1 102.883} C_DIS
LIN {X -0.224,Y -453.720,Z 352.560,A 0.000,B 0.000,C 90.000,E1 100.894} C_DIS
LIN {X -0.157,Y -474.499,Z 352.550,A 0.000,B 0.000,C 90.000,E1 99.029} C_DIS
LIN {X -0.167,Y -492.965,Z 352.542,A 0.000,B 0.000,C 90.000,E1 97.530} C_DIS
LIN {X 0.146,Y -496.539,Z 352.539,A 0.000,B 0.000,C 90.000,E1 97.068} C_DIS
LIN {X 0.051,Y -497.908,Z 352.538,A 0.000,B 0.000,C 90.000,E1 96.834} C_DIS
LIN {X -0.103,Y -498.919,Z 352.537,A 0.000,B 0.000,C 90.000,E1 96.606} C_DIS
LIN {X 0.172,Y -500.055,Z 352.534,A 0.000,B 0.000,C 90.000,E1 96.087} C_DIS
LIN {X -0.047,Y -500.167,Z 352.531,A 0.000,B 0.000,C 90.000,E1 95.625} C_DIS
LIN {X 0.238,Y -499.273,Z 352.529,A 0.000,B 0.000,C 90.000,E1 95.106} C_DIS
LIN {X 0.024,Y -497.213,Z 352.526,A 0.000,B 0.000,C 90.000,E1 94.645} C_DIS
LIN {X -0.232,Y -493.870,Z 352.523,A 0.000,B 0.000,C 90.000,E1 94.188} C_DIS
LIN {X -0.123,Y -488.346,Z 352.519,A 0.000,B 0.000,C 90.000,E1 93.440} C_DIS
LIN {X 0.099,Y -478.350,Z 352.512,A 0.000,B 0.000,C 90.000,E1 92.178} C_DIS
LIN {X 0.102,Y -454.908,Z 352.495,A 0.000,B 0.000,C 90.000,E1 89.141} C_DIS
LIN {X -0.027,Y -440.529,Z 352.484,A 0.000,B 0.000,C 90.000,E1 87.078} C_DIS
LIN {X -0.008,Y -422.455,Z 352.467,A 0.000,B 0.000,C 90.000,E1 84.147} C_DIS
LIN {X 0.007,Y -405.899,Z 352.451,A 0.000,B 0.000,C 90.000,E1 81.141} C_DIS
LIN {X 0.196,Y -395.670,Z 352.440,A 0.000,B 0.000,C 90.000,E1 79.162} C_DIS
LIN {X -0.132,Y -385.486,Z 352.429,A 0.000,B 0.000,C 90.000,E1 77.229} C_DIS
LIN {X -0.101,Y -373.852,Z 352.416,A 0.000,B 0.000,C 90.000,E1 74.921} C_DIS
LIN {X 0.098,Y -362.282,Z 352.403,A 0.000,B 0.000,C 90.000,E1 72.543} C_DIS
LIN {X -0.050,Y -352.080,Z 352.392,A 0.000,B 0.000,C 90.000,E1 70.477} C_DIS
LIN {X 0.072,Y -336.481,Z 352.373,A 0.000,B 0.000,C 90.000,E1 67.102} C_DIS
LIN {X 0.137,Y -324.763,Z 352.357,A 0.000,B 0.000,C 90.000,E1 64.280} C_DIS
LIN {X -0.048,Y -315.185,Z 352.343,A 0.000,B 0.000,C 90.000,E1 61.769} C_DIS
LIN {X -0.043,Y -302.758,Z 352.323,A 0.000,B 0.000,C 90.000,E1 58.201} C_DIS
LIN {X -0.043,Y -292.346,Z 352.305,A 0.000,B 0.000,C 90.000,E1 54.895} C_DIS
LIN {X -0.086,Y -282.705,Z 352.286,A 0.000,B 0.000,C 90.000,E1 51.537} C_DIS
LIN {X 0.056,Y -275.206,Z 352.271,A 0.000,B 0.000,C 90.000,E1 48.771} C_DIS
LIN {X 0.013,Y -269.513,Z 352.259,A 0.000,B 0.000,C 90.000,E1 46.701} C_DIS
LIN {X 0.148,Y -261.957,Z 352.244,A 0.000,B 0.000,C 90.000,E1 43.866} C_DIS
LIN {X -0.074,Y -254.373,Z 352.228,A 0.000,B 0.000,C 90.000,E1 41.067} C_DIS
LIN {X -0.101,Y -248.580,Z 352.216,A 0.000,B 0.000,C 90.000,E1 38.910} C_DIS
LIN {X -0.045,Y -242.650,Z 352.204,A 0.000,B 0.000,C 90.000,E1 36.710} C_DIS
LIN {X 0.141,Y -234.868,Z 352.187,A 0.000,B 0.000,C 90.000,E1 33.706} C_DIS
LIN {X -0.097,Y -225.542,Z 352.167,A 0.000,B 0.000,C 90.000,E1 30.001} C_DIS
LIN {X -0.042,Y -218.708,Z 352.150,A 0.000,B 0.000,C 90.000,E1 26.924} C_DIS
LIN {X -0.013,Y -210.991,Z 352.128,A 0.000,B 0.000,C 90.000,E1 23.025} C_DIS
LIN {X -0.008,Y -205.609,Z 352.110,A 0.000,B 0.000,C 90.000,E1 19.866} C_DIS
LIN {X 0.076,Y -199.875,Z 352.088,A 0.000,B 0.000,C 90.000,E1 15.843} C_DIS
LIN {X -0.031,Y -195.126,Z 352.066,A 0.000,B 0.000,C 90.000,E1 11.827} C_DIS
LIN {X 0.096,Y -191.506,Z 352.043,A 0.000,B 0.000,C 90.000,E1 7.701} C_DIS
LIN {X -0.082,Y -188.740,Z 352.015,A 0.000,B 0.000,C 90.000,E1 2.808} C_DIS
LIN {X -0.025,Y -189.620,Z 351.938,A 0.000,B 0.000,C 90.000,E1 348.757} C_DIS
LIN {X 0.016,Y -192.726,Z 351.910,A 0.000,B 0.000,C 90.000,E1 343.795} C_DIS
LIN {X 0.014,Y -196.527,Z 351.887,A 0.000,B 0.000,C 90.000,E1 339.699} C_DIS
LIN {X -0.079,Y -201.374,Z 351.865,A 0.000,B 0.000,C 90.000,E1 335.665} C_DIS
LIN {X -0.049,Y -207.290,Z 351.842,A 0.000,B 0.000,C 90.000,E1 331.641} C_DIS
LIN {X 0.017,Y -214.091,Z 351.820,A 0.000,B 0.000,C 90.000,E1 327.661} C_DIS
LIN {X 0.031,Y -220.134,Z 351.803,A 0.000,B 0.000,C 90.000,E1 324.529} C_DIS
LIN {X 0.024,Y -228.344,Z 351.782,A 0.000,B 0.000,C 90.000,E1 320.678} C_DIS
LIN {X 0.064,Y -235.754,Z 351.765,A 0.000,B 0.000,C 90.000,E1 317.634} C_DIS
LIN {X 0.108,Y -245.109,Z 351.746,A 0.000,B 0.000,C 90.000,E1 314.271} C_DIS
LIN {X 0.101,Y -255.773,Z 351.728,A 0.000,B 0.000,C 90.000,E1 310.987} C_DIS
LIN {X -0.077,Y -267.248,Z 351.710,A 0.000,B 0.000,C 90.000,E1 307.810} C_DIS
LIN {X -0.052,Y -279.772,Z 351.693,A 0.000,B 0.000,C 90.000,E1 304.659} C_DIS
LIN {X -0.051,Y -292.125,Z 351.677,A 0.000,B 0.000,C 90.000,E1 301.926} C_DIS
LIN {X -0.132,Y -309.351,Z 351.659,A 0.000,B 0.000,C 90.000,E1 298.615} C_DIS
LIN {X 0.097,Y -318.821,Z 351.650,A 0.000,B 0.000,C 90.000,E1 296.950} C_DIS
LIN {X -0.130,Y -339.843,Z 351.632,A 0.000,B 0.000,C 90.000,E1 293.823} C_DIS
LIN {X -0.070,Y -355.503,Z 351.620,A 0.000,B 0.000,C 90.000,E1 291.663} C_DIS
LIN {X -0.116,Y -371.770,Z 351.609,A 0.000,B 0.000,C 90.000,E1 289.577} C_DIS
LIN {X 0.125,Y -391.837,Z 351.596,A 0.000,B 0.000,C 90.000,E1 287.221} C_DIS
LIN {X 0.154,Y -407.201,Z 351.587,A 0.000,B 0.000,C 90.000,E1 285.552} C_DIS
LIN {X -0.187,Y -419.536,Z 351.579,A 0.000,B 0.000,C 90.000,E1 284.300} C_DIS
LIN {X 0.230,Y -429.466,Z 351.573,A 0.000,B 0.000,C 90.000,E1 283.175} C_DIS
LIN {X 0.108,Y -438.857,Z 351.567,A 0.000,B 0.000,C 90.000,E1 282.119} C_DIS
LIN {X -0.216,Y -445.372,Z 351.563,A 0.000,B 0.000,C 90.000,E1 281.366} C_DIS
LIN {X -0.159,Y -453.227,Z 351.557,A 0.000,B 0.000,C 90.000,E1 280.310} C_DIS
LIN {X -0.092,Y -460.567,Z 351.551,A 0.000,B 0.000,C 90.000,E1 279.265} C_DIS
LIN {X 0.064,Y -467.276,Z 351.546,A 0.000,B 0.000,C 90.000,E1 278.219} C_DIS
LIN {X -0.234,Y -473.502,Z 351.540,A 0.000,B 0.000,C 90.000,E1 277.239} C_DIS
LIN {X 0.012,Y -479.045,Z 351.534,A 0.000,B 0.000,C 90.000,E1 276.201} C_DIS
LIN {X -0.021,Y -482.641,Z 351.530,A 0.000,B 0.000,C 90.000,E1 275.454} C_DIS
LIN {X 0.153,Y -484.682,Z 351.528,A 0.000,B 0.000,C 90.000,E1 274.935} C_DIS
LIN {X -0.153,Y -486.288,Z 351.525,A 0.000,B 0.000,C 90.000,E1 274.473} C_DIS
LIN {X 0.034,Y -487.472,Z 351.522,A 0.000,B 0.000,C 90.000,E1 273.955} C_DIS
LIN {X 0.199,Y -488.305,Z 351.519,A 0.000,B 0.000,C 90.000,E1 273.440} C_DIS
LIN {X -0.087,Y -488.747,Z 351.517,A 0.000,B 0.000,C 90.000,E1 272.980} C_DIS
LIN {X 0.093,Y -488.895,Z 351.514,A 0.000,B 0.000,C 90.000,E1 272.465} C_DIS
LIN {X -0.209,Y -488.763,Z 351.511,A 0.000,B 0.000,C 90.000,E1 272.007} C_DIS
LIN {X -0.007,Y -488.342,Z 351.508,A 0.000,B 0.000,C 90.000,E1 271.489} C_DIS
LIN {X 0.179,Y -487.660,Z 351.506,A 0.000,B 0.000,C 90.000,E1 270.974} C_DIS
LIN {X -0.123,Y -486.648,Z 351.503,A 0.000,B 0.000,C 90.000,E1 270.516} C_DIS
LIN {X 0.058,Y -485.282,Z 351.500,A 0.000,B 0.000,C 90.000,E1 270.000} C_DIS
LIN {X 0.074,Y -482.240,Z 351.496,A 0.000,B 0.000,C 90.000,E1 269.255} C_DIS
LIN {X 0.230,Y -479.503,Z 351.493,A 0.000,B 0.000,C 90.000,E1 268.740} C_DIS
LIN {X -0.111,Y -475.907,Z 351.490,A 0.000,B 0.000,C 90.000,E1 268.282} C_DIS
LIN {X 0.023,Y -471.277,Z 351.488,A 0.000,B 0.000,C 90.000,E1 267.764} C_DIS
LIN {X -0.158,Y -468.534,Z 351.486,A 0.000,B 0.000,C 90.000,E1 267.535} C_DIS
LIN {X -0.199,Y -465.641,Z 351.485,A 0.000,B 0.000,C 90.000,E1 267.306} C_DIS
LIN {X 0.220,Y -462.327,Z 351.484,A 0.000,B 0.000,C 90.000,E1 267.020} C_DIS
LIN {X 0.046,Y -459.168,Z 351.483,A 0.000,B 0.000,C 90.000,E1 266.846} C_DIS
LIN {X -0.149,Y -455.475,Z 351.481,A 0.000,B 0.000,C 90.000,E1 266.674} C_DIS
LIN {X -0.030,Y -452.029,Z 351.481,A 0.000,B 0.000,C 90.000,E1 266.502} C_DIS
LIN {X 0.063,Y -444.307,Z 351.479,A 0.000,B 0.000,C 90.000,E1 266.216} C_DIS
LIN {X -0.185,Y -436.156,Z 351.478,A 0.000,B 0.000,C 90.000,E1 266.045} C_DIS
LIN {X 0.044,Y -427.258,Z 351.477,A 0.000,B 0.000,C 90.000,E1 265.869} C_DIS
LIN {X -0.026,Y -417.653,Z 351.477,A 0.000,B 0.000,C 90.000,E1 265.812} C_DIS
LIN {X -0.036,Y -180.913,Z 351.477,A 0.000,B 0.000,C 90.000,E1 265.812} C_DIS
LIN {X 0.058,Y -180.839,Z 351.472,A 0.000,B 0.000,C 90.000,E1 264.894} C_DIS
LIN {X -0.039,Y -178.947,Z 351.444,A 0.000,B 0.000,C 90.000,E1 259.859} C_DIS
LIN {X 0.057,Y -176.402,Z 351.420,A 0.000,B 0.000,C 90.000,E1 255.589} C_DIS
LIN {X -0.050,Y -175.508,Z 351.411,A 0.000,B 0.000,C 90.000,E1 253.921} C_DIS
LIN {X 0.012,Y -172.248,Z 351.387,A 0.000,B 0.000,C 90.000,E1 249.625} C_DIS
LIN {X -0.009,Y -171.726,Z 351.382,A 0.000,B 0.000,C 90.000,E1 248.773} C_DIS
LIN {X 0.000,Y -167.322,Z 351.353,A 0.000,B 0.000,C 90.000,E1 243.589} C_DIS
LIN {X -0.068,Y -166.706,Z 351.348,A 0.000,B 0.000,C 90.000,E1 242.743} C_DIS
LIN {X 0.070,Y -162.686,Z 351.324,A 0.000,B 0.000,C 90.000,E1 238.329} C_DIS
LIN {X 0.043,Y -161.376,Z 351.314,A 0.000,B 0.000,C 90.000,E1 236.580} C_DIS
LIN {X -0.049,Y -157.369,Z 351.290,A 0.000,B 0.000,C 90.000,E1 232.190} C_DIS
LIN {X -0.014,Y -155.361,Z 351.275,A 0.000,B 0.000,C 90.000,E1 229.504} C_DIS
LIN {X 0.033,Y -151.703,Z 351.250,A 0.000,B 0.000,C 90.000,E1 225.000} C_DIS
LIN {X -0.029,Y -150.564,Z 351.240,A 0.000,B 0.000,C 90.000,E1 223.218} C_DIS
LIN {X -0.002,Y -147.291,Z 351.215,A 0.000,B 0.000,C 90.000,E1 218.669} C_DIS
LIN {X -0.034,Y -145.320,Z 351.195,A 0.000,B 0.000,C 90.000,E1 215.025} C_DIS
LIN {X 0.005,Y -142.406,Z 351.164,A 0.000,B 0.000,C 90.000,E1 209.489} C_DIS
LIN {X -0.068,Y -141.390,Z 351.148,A 0.000,B 0.000,C 90.000,E1 206.744} C_DIS
LIN {X -0.080,Y -139.351,Z 351.112,A 0.000,B 0.000,C 90.000,E1 200.248} C_DIS
LIN {X 0.040,Y -138.790,Z 351.097,A 0.000,B 0.000,C 90.000,E1 197.402} C_DIS
LIN {X -0.037,Y -138.345,Z 351.055,A 0.000,B 0.000,C 90.000,E1 189.962} C_DIS
LIN {X -0.020,Y -139.381,Z 351.009,A 0.000,B 0.000,C 90.000,E1 181.547} C_DIS
LIN {X 0.034,Y -141.275,Z 350.972,A 0.000,B 0.000,C 90.000,E1 175.008} C_DIS
LIN {X -0.009,Y -142.640,Z 350.957,A 0.000,B 0.000,C 90.000,E1 172.243} C_DIS
LIN {X -0.057,Y -144.972,Z 350.931,A 0.000,B 0.000,C 90.000,E1 167.645} C_DIS
LIN {X -0.067,Y -147.599,Z 350.911,A 0.000,B 0.000,C 90.000,E1 163.976} C_DIS
LIN {X 0.013,Y -150.218,Z 350.891,A 0.000,B 0.000,C 90.000,E1 160.296} C_DIS
LIN {X 0.029,Y -153.606,Z 350.870,A 0.000,B 0.000,C 90.000,E1 156.666} C_DIS
LIN {X 0.018,Y -157.021,Z 350.850,A 0.000,B 0.000,C 90.000,E1 153.076} C_DIS
LIN {X -0.051,Y -161.143,Z 350.831,A 0.000,B 0.000,C 90.000,E1 149.537} C_DIS
LIN {X 0.032,Y -163.241,Z 350.821,A 0.000,B 0.000,C 90.000,E1 147.740} C_DIS
LIN {X -0.005,Y -167.676,Z 350.801,A 0.000,B 0.000,C 90.000,E1 144.242} C_DIS
LIN {X 0.045,Y -171.499,Z 350.787,A 0.000,B 0.000,C 90.000,E1 141.618} C_DIS
LIN {X 0.089,Y -176.432,Z 350.768,A 0.000,B 0.000,C 90.000,E1 138.162} C_DIS
LIN {X -0.040,Y -180.728,Z 350.754,A 0.000,B 0.000,C 90.000,E1 135.648} C_DIS
LIN {X -0.059,Y -186.132,Z 350.735,A 0.000,B 0.000,C 90.000,E1 132.285} C_DIS
LIN {X -0.003,Y -190.770,Z 350.721,A 0.000,B 0.000,C 90.000,E1 129.769} C_DIS
LIN {X 0.064,Y -196.525,Z 350.703,A 0.000,B 0.000,C 90.000,E1 126.457} C_DIS
LIN {X 0.087,Y -200.190,Z 350.692,A 0.000,B 0.000,C 90.000,E1 124.612} C_DIS
LIN {X 0.095,Y -300.501,Z 350.692,A 0.000,B 0.000,C 90.000,E1 124.612} C_DIS
LIN {X -0.175,Y -302.931,Z 350.692,A 0.000,B 0.000,C 90.000,E1 124.612} C_DIS
LIN {X -0.101,Y -307.719,Z 350.691,A 0.000,B 0.000,C 90.000,E1 124.326} C_DIS
LIN {X -0.025,Y -310.441,Z 350.689,A 0.000,B 0.000,C 90.000,E1 124.040} C_DIS
LIN {X -0.150,Y -314.137,Z 350.686,A 0.000,B 0.000,C 90.000,E1 123.499} C_DIS
LIN {X -0.101,Y -315.626,Z 350.684,A 0.000,B 0.000,C 90.000,E1 123.166} C_DIS
LIN {X 0.077,Y -328.581,Z 350.665,A 0.000,B 0.000,C 90.000,E1 119.617} C_DIS
LIN {X -0.040,Y -340.632,Z 350.649,A 0.000,B 0.000,C 90.000,E1 116.821} C_DIS
LIN {X 0.159,Y -352.595,Z 350.635,A 0.000,B 0.000,C 90.000,E1 114.335} C_DIS
LIN {X -0.101,Y -365.820,Z 350.622,A 0.000,B 0.000,C 90.000,E1 111.972} C_DIS
LIN {X -0.179,Y -380.408,Z 350.609,A 0.000,B 0.000,C 90.000,E1 109.631} C_DIS
LIN {X 0.214,Y -396.466,Z 350.596,A 0.000,B 0.000,C 90.000,E1 107.275} C_DIS
LIN {X 0.019,Y -414.111,Z 350.584,A 0.000,B 0.000,C 90.000,E1 105.064} C_DIS
LIN {X 0.069,Y -433.431,Z 350.572,A 0.000,B 0.000,C 90.000,E1 102.883} C_DIS
LIN {X -0.212,Y -453.675,Z 350.560,A 0.000,B 0.000,C 90.000,E1 100.894} C_DIS
LIN {X -0.147,Y -474.454,Z 350.550,A 0.000,B 0.000,C 90.000,E1 99.029} C_DIS
LIN {X -0.159,Y -492.953,Z 350.542,A 0.000,B 0.000,C 90.000,E1 97.530} C_DIS
LIN {X 0.186,Y -496.586,Z 350.539,A 0.000,B 0.000,C 90.000,E1 97.068} C_DIS
LIN {X 0.092,Y -497.992,Z 350.538,A 0.000,B 0.000,C 90.000,E1 96.834} C_DIS
LIN {X -0.063,Y -499.033,Z 350.537,A 0.000,B 0.000,C 90.000,E1 96.606} C_DIS
LIN {X 0.212,Y -500.218,Z 350.534,A 0.000,B 0.000,C 90.000,E1 96.087} C_DIS
LIN {X -0.005,Y -500.374,Z 350.531,A 0.000,B 0.000,C 90.000,E1 95.625} C_DIS
LIN {X -0.217,Y -499.526,Z 350.529,A 0.000,B 0.000,C 90.000,E1 95.163} C_DIS
LIN {X 0.067,Y -497.524,Z 350.526,A 0.000,B 0.000,C 90.000,E1 94.645} C_DIS
LIN {X -0.187,Y -494.204,Z 350.523,A 0.000,B 0.000,C 90.000,E1 94.188} C_DIS
LIN {X -0.217,Y -486.734,Z 350.518,A 0.000,B 0.000,C 90.000,E1 93.212} C_DIS
LIN {X -0.175,Y -474.664,Z 350.509,A 0.000,B 0.000,C 90.000,E1 91.718} C_DIS
LIN {X 0.159,Y -451.481,Z 350.492,A 0.000,B 0.000,C 90.000,E1 88.625} C_DIS
LIN {X -0.134,Y -434.039,Z 350.478,A 0.000,B 0.000,C 90.000,E1 86.045} C_DIS
LIN {X -0.132,Y -415.078,Z 350.460,A 0.000,B 0.000,C 90.000,E1 82.818} C_DIS
LIN {X 0.024,Y -400.340,Z 350.445,A 0.000,B 0.000,C 90.000,E1 80.038} C_DIS
LIN {X -0.152,Y -388.704,Z 350.432,A 0.000,B 0.000,C 90.000,E1 77.813} C_DIS
LIN {X -0.134,Y -377.056,Z 350.419,A 0.000,B 0.000,C 90.000,E1 75.519} C_DIS
LIN {X 0.143,Y -365.481,Z 350.406,A 0.000,B 0.000,C 90.000,E1 73.142} C_DIS
LIN {X -0.054,Y -355.276,Z 350.395,A 0.000,B 0.000,C 90.000,E1 71.094} C_DIS
LIN {X 0.127,Y -343.668,Z 350.381,A 0.000,B 0.000,C 90.000,E1 68.646} C_DIS
LIN {X -0.118,Y -327.486,Z 350.361,A 0.000,B 0.000,C 90.000,E1 64.973} C_DIS
LIN {X -0.013,Y -316.627,Z 350.345,A 0.000,B 0.000,C 90.000,E1 62.103} C_DIS
LIN {X 0.032,Y -304.087,Z 350.325,A 0.000,B 0.000,C 90.000,E1 58.535} C_DIS
LIN {X 0.071,Y -292.594,Z 350.305,A 0.000,B 0.000,C 90.000,E1 54.895} C_DIS
LIN {X 0.032,Y -282.929,Z 350.286,A 0.000,B 0.000,C 90.000,E1 51.537} C_DIS
LIN {X -0.005,Y -275.429,Z 350.271,A 0.000,B 0.000,C 90.000,E1 48.809} C_DIS
LIN {X -0.061,Y -269.744,Z 350.260,A 0.000,B 0.000,C 90.000,E1 46.743} C_DIS
LIN {X -0.098,Y -262.187,Z 350.244,A 0.000,B 0.000,C 90.000,E1 43.947} C_DIS
LIN {X 0.167,Y -256.507,Z 350.232,A 0.000,B 0.000,C 90.000,E1 41.757} C_DIS
LIN {X -0.017,Y -250.784,Z 350.220,A 0.000,B 0.000,C 90.000,E1 39.644} C_DIS
LIN {X 0.079,Y -244.901,Z 350.208,A 0.000,B 0.000,C 90.000,E1 37.443} C_DIS
LIN {X -0.066,Y -237.034,Z 350.192,A 0.000,B 0.000,C 90.000,E1 34.532} C_DIS
LIN {X -0.113,Y -227.549,Z 350.171,A 0.000,B 0.000,C 90.000,E1 30.797} C_DIS
LIN {X -0.004,Y -220.547,Z 350.154,A 0.000,B 0.000,C 90.000,E1 27.719} C_DIS
LIN {X 0.069,Y -212.609,Z 350.132,A 0.000,B 0.000,C 90.000,E1 23.823} C_DIS
LIN {X 0.037,Y -207.007,Z 350.115,A 0.000,B 0.000,C 90.000,E1 20.684} C_DIS
LIN {X 0.105,Y -201.051,Z 350.093,A 0.000,B 0.000,C 90.000,E1 16.677} C_DIS
LIN {X 0.079,Y -196.122,Z 350.070,A 0.000,B 0.000,C 90.000,E1 12.647} C_DIS
LIN {X 0.075,Y -192.217,Z 350.048,A 0.000,B 0.000,C 90.000,E1 8.568} C_DIS
LIN {X -0.059,Y -189.183,Z 350.020,A 0.000,B 0.000,C 90.000,E1 3.669} C_DIS
LIN {X 0.022,Y -187.936,Z 349.970,A 0.000,B 0.000,C 90.000,E1 354.546} C_DIS
LIN {X -0.043,Y -190.040,Z 349.933,A 0.000,B 0.000,C 90.000,E1 347.937} C_DIS
LIN {X 0.062,Y -193.413,Z 349.905,A 0.000,B 0.000,C 90.000,E1 342.960} C_DIS
LIN {X -0.041,Y -197.400,Z 349.883,A 0.000,B 0.000,C 90.000,E1 338.901} C_DIS
LIN {X -0.027,Y -202.438,Z 349.860,A 0.000,B 0.000,C 90.000,E1 334.845} C_DIS
LIN {X -0.051,Y -208.519,Z 349.838,A 0.000,B 0.000,C 90.000,E1 330.845} C_DIS
LIN {X -0.129,Y -215.488,Z 349.816,A 0.000,B 0.000,C 90.000,E1 326.914} C_DIS
LIN {X -0.063,Y -223.290,Z 349.794,A 0.000,B 0.000,C 90.000,E1 323.004} C_DIS
LIN {X 0.050,Y -230.035,Z 349.777,A 0.000,B 0.000,C 90.000,E1 319.908} C_DIS
LIN {X -0.067,Y -238.669,Z 349.758,A 0.000,B 0.000,C 90.000,E1 316.539} C_DIS
LIN {X 0.071,Y -248.489,Z 349.740,A 0.000,B 0.000,C 90.000,E1 313.176} C_DIS
LIN {X -0.005,Y -259.486,Z 349.722,A 0.000,B 0.000,C 90.000,E1 309.930} C_DIS
LIN {X -0.038,Y -271.287,Z 349.704,A 0.000,B 0.000,C 90.000,E1 306.744} C_DIS
LIN {X -0.049,Y -284.279,Z 349.687,A 0.000,B 0.000,C 90.000,E1 303.627} C_DIS
LIN {X -0.081,Y -295.538,Z 349.674,A 0.000,B 0.000,C 90.000,E1 301.258} C_DIS
LIN {X -0.200,Y -313.206,Z 349.655,A 0.000,B 0.000,C 90.000,E1 297.975} C_DIS
LIN {X 0.096,Y -323.107,Z 349.646,A 0.000,B 0.000,C 90.000,E1 296.309} C_DIS
LIN {X -0.135,Y -342.335,Z 349.631,A 0.000,B 0.000,C 90.000,E1 293.515} C_DIS
LIN {X -0.009,Y -358.034,Z 349.619,A 0.000,B 0.000,C 90.000,E1 291.354} C_DIS
LIN {X -0.005,Y -374.491,Z 349.607,A 0.000,B 0.000,C 90.000,E1 289.268} C_DIS
LIN {X -0.099,Y -394.722,Z 349.594,A 0.000,B 0.000,C 90.000,E1 286.968} C_DIS
LIN {X 0.081,Y -409.953,Z 349.585,A 0.000,B 0.000,C 90.000,E1 285.300} C_DIS
LIN {X -0.130,Y -422.420,Z 349.578,A 0.000,B 0.000,C 90.000,E1 284.008} C_DIS
LIN {X 0.079,Y -429.825,Z 349.573,A 0.000,B 0.000,C 90.000,E1 283.175} C_DIS
LIN {X 0.195,Y -436.873,Z 349.569,A 0.000,B 0.000,C 90.000,E1 282.355} C_DIS
LIN {X -0.062,Y -443.449,Z 349.564,A 0.000,B 0.000,C 90.000,E1 281.591} C_DIS
LIN {X 0.093,Y -449.533,Z 349.560,A 0.000,B 0.000,C 90.000,E1 280.782} C_DIS
LIN {X 0.201,Y -457.076,Z 349.554,A 0.000,B 0.000,C 90.000,E1 279.726} C_DIS
LIN {X -0.212,Y -464.056,Z 349.548,A 0.000,B 0.000,C 90.000,E1 278.746} C_DIS
LIN {X -0.014,Y -470.522,Z 349.543,A 0.000,B 0.000,C 90.000,E1 277.701} C_DIS
LIN {X 0.199,Y -476.368,Z 349.537,A 0.000,B 0.000,C 90.000,E1 276.663} C_DIS
LIN {X 0.193,Y -480.289,Z 349.533,A 0.000,B 0.000,C 90.000,E1 275.910} C_DIS
LIN {X -0.131,Y -482.633,Z 349.530,A 0.000,B 0.000,C 90.000,E1 275.448} C_DIS
LIN {X -0.004,Y -484.623,Z 349.527,A 0.000,B 0.000,C 90.000,E1 274.935} C_DIS
LIN {X 0.175,Y -486.227,Z 349.525,A 0.000,B 0.000,C 90.000,E1 274.416} C_DIS
LIN {X -0.123,Y -487.402,Z 349.522,A 0.000,B 0.000,C 90.000,E1 273.955} C_DIS
LIN {X 0.041,Y -488.206,Z 349.519,A 0.000,B 0.000,C 90.000,E1 273.440} C_DIS
LIN {X 0.242,Y -488.616,Z 349.516,A 0.000,B 0.000,C 90.000,E1 272.922} C_DIS
LIN {X -0.067,Y -488.743,Z 349.514,A 0.000,B 0.000,C 90.000,E1 272.465} C_DIS
LIN {X 0.120,Y -488.603,Z 349.511,A 0.000,B 0.000,C 90.000,E1 271.949} C_DIS
LIN {X -0.167,Y -488.181,Z 349.508,A 0.000,B 0.000,C 90.000,E1 271.489} C_DIS
LIN {X 0.018,Y -487.501,Z 349.505,A 0.000,B 0.000,C 90.000,E1 270.974} C_DIS
LIN {X 0.201,Y -486.510,Z 349.503,A 0.000,B 0.000,C 90.000,E1 270.458} C_DIS
LIN {X -0.104,Y -485.082,Z 349.500,A 0.000,B 0.000,C 90.000,E1 270.000} C_DIS
LIN {X 0.070,Y -483.253,Z 349.497,A 0.000,B 0.000,C 90.000,E1 269.484} C_DIS
LIN {X 0.233,Y -480.852,Z 349.494,A 0.000,B 0.000,C 90.000,E1 268.969} C_DIS
LIN {X -0.100,Y -477.653,Z 349.492,A 0.000,B 0.000,C 90.000,E1 268.511} C_DIS
LIN {X 0.202,Y -475.733,Z 349.490,A 0.000,B 0.000,C 90.000,E1 268.224} C_DIS
LIN {X -0.139,Y -471.079,Z 349.487,A 0.000,B 0.000,C 90.000,E1 267.764} C_DIS
LIN {X 0.149,Y -468.308,Z 349.486,A 0.000,B 0.000,C 90.000,E1 267.478} C_DIS
LIN {X 0.085,Y -462.105,Z 349.483,A 0.000,B 0.000,C 90.000,E1 267.020} C_DIS
LIN {X -0.093,Y -458.954,Z 349.482,A 0.000,B 0.000,C 90.000,E1 266.846} C_DIS
LIN {X 0.161,Y -455.239,Z 349.481,A 0.000,B 0.000,C 90.000,E1 266.617} C_DIS
LIN {X -0.048,Y -447.725,Z 349.480,A 0.000,B 0.000,C 90.000,E1 266.331} C_DIS
LIN {X -0.125,Y -439.592,Z 349.478,A 0.000,B 0.000,C 90.000,E1 266.102} C_DIS
LIN {X -0.083,Y -430.960,Z 349.477,A 0.000,B 0.000,C 90.000,E1 265.927} C_DIS
LIN {X 0.131,Y -423.984,Z 349.477,A 0.000,B 0.000,C 90.000,E1 265.812} C_DIS
LIN {X -0.129,Y -415.505,Z 349.477,A 0.000,B 0.000,C 90.000,E1 265.812} C_DIS
LIN {X -0.079,Y -180.913,Z 349.477,A 0.000,B 0.000,C 90.000,E1 265.812} C_DIS
LIN {X 0.025,Y -180.836,Z 349.472,A 0.000,B 0.000,C 90.000,E1 264.894} C_DIS
LIN {X -0.072,Y -178.944,Z 349.444,A 0.000,B 0.000,C 90.000,E1 259.859} C_DIS
LIN {X -0.028,Y -175.995,Z 349.415,A 0.000,B 0.000,C 90.000,E1 254.755} C_DIS
LIN {X -0.083,Y -175.500,Z 349.411,A 0.000,B 0.000,C 90.000,E1 253.921} C_DIS
LIN {X -0.020,Y -172.241,Z 349.387,A 0.000,B 0.000,C 90.000,E1 249.625} C_DIS
LIN {X -0.041,Y -171.719,Z 349.382,A 0.000,B 0.000,C 90.000,E1 248.773} C_DIS
LIN {X -0.032,Y -167.315,Z 349.353,A 0.000,B 0.000,C 90.000,E1 243.589} C_DIS
LIN {X 0.049,Y -166.697,Z 349.348,A 0.000,B 0.000,C 90.000,E1 242.692} C_DIS
LIN {X 0.040,Y -162.677,Z 349.324,A 0.000,B 0.000,C 90.000,E1 238.329} C_DIS
LIN {X 0.013,Y -161.367,Z 349.314,A 0.000,B 0.000,C 90.000,E1 236.580} C_DIS
LIN {X -0.078,Y -157.360,Z 349.290,A 0.000,B 0.000,C 90.000,E1 232.190} C_DIS
LIN {X 0.075,Y -155.350,Z 349.275,A 0.000,B 0.000,C 90.000,E1 229.461} C_DIS
LIN {X 0.004,Y -151.696,Z 349.250,A 0.000,B 0.000,C 90.000,E1 225.000} C_DIS
LIN {X 0.052,Y -150.558,Z 349.240,A 0.000,B 0.000,C 90.000,E1 223.176} C_DIS
LIN {X -0.032,Y -147.284,Z 349.215,A 0.000,B 0.000,C 90.000,E1 218.669} C_DIS
LIN {X -0.063,Y -145.313,Z 349.194,A 0.000,B 0.000,C 90.000,E1 215.025} C_DIS
LIN {X 0.048,Y -142.402,Z 349.164,A 0.000,B 0.000,C 90.000,E1 209.461} C_DIS
LIN {X 0.031,Y -141.384,Z 349.148,A 0.000,B 0.000,C 90.000,E1 206.693} C_DIS
LIN {X 0.023,Y -139.349,Z 349.112,A 0.000,B 0.000,C 90.000,E1 200.194} C_DIS
LIN {X 0.013,Y -138.788,Z 349.097,A 0.000,B 0.000,C 90.000,E1 197.402} C_DIS
LIN {X -0.065,Y -138.344,Z 349.055,A 0.000,B 0.000,C 90.000,E1 189.962} C_DIS
LIN {X -0.048,Y -139.384,Z 349.008,A 0.000,B 0.000,C 90.000,E1 181.547} C_DIS
LIN {X 0.006,Y -141.279,Z 348.972,A 0.000,B 0.000,C 90.000,E1 175.008} C_DIS
LIN {X -0.036,Y -142.644,Z 348.957,A 0.000,B 0.000,C 90.000,E1 172.243} C_DIS
LIN {X 0.056,Y -144.979,Z 348.931,A 0.000,B 0.000,C 90.000,E1 167.589} C_DIS
LIN {X 0.045,Y -147.606,Z 348.911,A 0.000,B 0.000,C 90.000,E1 163.921} C_DIS
LIN {X -0.016,Y -150.227,Z 348.891,A 0.000,B 0.000,C 90.000,E1 160.296} C_DIS
LIN {X -0.001,Y -153.617,Z 348.870,A 0.000,B 0.000,C 90.000,E1 156.666} C_DIS
LIN {X -0.012,Y -157.033,Z 348.850,A 0.000,B 0.000,C 90.000,E1 153.076} C_DIS
LIN {X -0.082,Y -161.156,Z 348.831,A 0.000,B 0.000,C 90.000,E1 149.537} C_DIS
LIN {X 0.001,Y -163.254,Z 348.821,A 0.000,B 0.000,C 90.000,E1 147.740} C_DIS
LIN {X 0.100,Y -167.691,Z 348.801,A 0.000,B 0.000,C 90.000,E1 144.196} C_DIS
LIN {X 0.013,Y -171.512,Z 348.787,A 0.000,B 0.000,C 90.000,E1 141.618} C_DIS
LIN {X 0.056,Y -176.448,Z 348.768,A 0.000,B 0.000,C 90.000,E1 138.162} C_DIS
LIN {X -0.073,Y -180.745,Z 348.753,A 0.000,B 0.000,C 90.000,E1 135.648} C_DIS
LIN {X 0.045,Y -186.150,Z 348.735,A 0.000,B 0.000,C 90.000,E1 132.243} C_DIS
LIN {X -0.036,Y -190.788,Z 348.721,A 0.000,B 0.000,C 90.000,E1 129.769} C_DIS
LIN {X 0.030,Y -196.544,Z 348.703,A 0.000,B 0.000,C 90.000,E1 126.457} C_DIS
LIN {X -0.052,Y -200.274,Z 348.692,A 0.000,B 0.000,C 90.000,E1 124.612} C_DIS
LIN {X -0.128,Y -300.402,Z 348.692,A 0.000,B 0.000,C 90.000,E1 124.612} C_DIS
LIN {X 0.021,Y -301.758,Z 348.692,A 0.000,B 0.000,C 90.000,E1 124.565} C_DIS
LIN {X 0.099,Y -307.415,Z 348.691,A 0.000,B 0.000,C 90.000,E1 124.278} C_DIS
LIN {X -0.080,Y -310.270,Z 348.689,A 0.000,B 0.000,C 90.000,E1 124.040} C_DIS
LIN {X -0.090,Y -313.972,Z 348.686,A 0.000,B 0.000,C 90.000,E1 123.499} C_DIS
LIN {X -0.041,Y -315.526,Z 348.684,A 0.000,B 0.000,C 90.000,E1 123.166} C_DIS
LIN {X -0.149,Y -328.519,Z 348.665,A 0.000,B 0.000,C 90.000,E1 119.667} C_DIS
LIN {X 0.020,Y -340.564,Z 348.649,A 0.000,B 0.000,C 90.000,E1 116.821} C_DIS
LIN {X -0.103,Y -352.521,Z 348.635,A 0.000,B 0.000,C 90.000,E1 114.387} C_DIS
LIN {X -0.040,Y -365.741,Z 348.622,A 0.000,B 0.000,C 90.000,E1 111.972} C_DIS
LIN {X -0.119,Y -380.323,Z 348.609,A 0.000,B 0.000,C 90.000,E1 109.631} C_DIS
LIN {X -0.102,Y -396.374,Z 348.596,A 0.000,B 0.000,C 90.000,E1 107.330} C_DIS
LIN {X 0.080,Y -414.012,Z 348.584,A 0.000,B 0.000,C 90.000,E1 105.064} C_DIS
LIN {X 0.129,Y -433.327,Z 348.572,A 0.000,B 0.000,C 90.000,E1 102.883} C_DIS
LIN {X -0.155,Y -453.569,Z 348.560,A 0.000,B 0.000,C 90.000,E1 100.894} C_DIS
LIN {X -0.093,Y -474.346,Z 348.550,A 0.000,B 0.000,C 90.000,E1 99.029} C_DIS
LIN {X -0.107,Y -492.879,Z 348.542,A 0.000,B 0.000,C 90.000,E1 97.530} C_DIS
LIN {X -0.222,Y -496.599,Z 348.539,A 0.000,B 0.000,C 90.000,E1 97.125} C_DIS
LIN {X 0.176,Y -498.052,Z 348.538,A 0.000,B 0.000,C 90.000,E1 96.834} C_DIS
LIN {X 0.021,Y -499.130,Z 348.537,A 0.000,B 0.000,C 90.000,E1 96.606} C_DIS
LIN {X -0.200,Y -500.375,Z 348.534,A 0.000,B 0.000,C 90.000,E1 96.144} C_DIS
LIN {X 0.081,Y -500.583,Z 348.531,A 0.000,B 0.000,C 90.000,E1 95.625} C_DIS
LIN {X -0.131,Y -499.789,Z 348.529,A 0.000,B 0.000,C 90.000,E1 95.163} C_DIS
LIN {X 0.155,Y -497.855,Z 348.526,A 0.000,B 0.000,C 90.000,E1 94.645} C_DIS
LIN {X -0.100,Y -494.609,Z 348.523,A 0.000,B 0.000,C 90.000,E1 94.188} C_DIS
LIN {X -0.126,Y -487.131,Z 348.518,A 0.000,B 0.000,C 90.000,E1 93.212} C_DIS
LIN {X -0.079,Y -475.059,Z 348.509,A 0.000,B 0.000,C 90.000,E1 91.718} C_DIS
LIN {X 0.037,Y -453.687,Z 348.494,A 0.000,B 0.000,C 90.000,E1 88.912} C_DIS
LIN {X -0.095,Y -439.429,Z 348.482,A 0.000,B 0.000,C 90.000,E1 86.846} C_DIS
LIN {X 0.174,Y -423.055,Z 348.468,A 0.000,B 0.000,C 90.000,E1 84.147} C_DIS
LIN {X 0.087,Y -407.921,Z 348.452,A 0.000,B 0.000,C 90.000,E1 81.432} C_DIS
LIN {X 0.008,Y -396.299,Z 348.440,A 0.000,B 0.000,C 90.000,E1 79.218} C_DIS
LIN {X 0.076,Y -386.101,Z 348.429,A 0.000,B 0.000,C 90.000,E1 77.229} C_DIS
LIN {X 0.019,Y -374.475,Z 348.416,A 0.000,B 0.000,C 90.000,E1 74.936} C_DIS
LIN {X -0.022,Y -362.911,Z 348.403,A 0.000,B 0.000,C 90.000,E1 72.598} C_DIS
LIN {X 0.064,Y -352.662,Z 348.392,A 0.000,B 0.000,C 90.000,E1 70.496} C_DIS
LIN {X -0.129,Y -336.971,Z 348.373,A 0.000,B 0.000,C 90.000,E1 67.177} C_DIS
LIN {X 0.089,Y -325.270,Z 348.357,A 0.000,B 0.000,C 90.000,E1 64.332} C_DIS
LIN {X -0.151,Y -314.537,Z 348.342,A 0.000,B 0.000,C 90.000,E1 61.513} C_DIS
LIN {X -0.043,Y -303.267,Z 348.324,A 0.000,B 0.000,C 90.000,E1 58.250} C_DIS
LIN {X -0.187,Y -292.864,Z 348.305,A 0.000,B 0.000,C 90.000,E1 54.975} C_DIS
LIN {X -0.037,Y -283.175,Z 348.287,A 0.000,B 0.000,C 90.000,E1 51.582} C_DIS
LIN {X -0.057,Y -275.688,Z 348.271,A 0.000,B 0.000,C 90.000,E1 48.852} C_DIS
LIN {X 0.061,Y -268.088,Z 348.256,A 0.000,B 0.000,C 90.000,E1 46.053} C_DIS
LIN {X -0.019,Y -260.570,Z 348.240,A 0.000,B 0.000,C 90.000,E1 43.257} C_DIS
LIN {X 0.088,Y -252.963,Z 348.224,A 0.000,B 0.000,C 90.000,E1 40.378} C_DIS
LIN {X 0.028,Y -247.133,Z 348.212,A 0.000,B 0.000,C 90.000,E1 38.222} C_DIS
LIN {X -0.063,Y -239.241,Z 348.196,A 0.000,B 0.000,C 90.000,E1 35.311} C_DIS
LIN {X 0.085,Y -229.658,Z 348.175,A 0.000,B 0.000,C 90.000,E1 31.544} C_DIS
LIN {X -0.039,Y -222.463,Z 348.158,A 0.000,B 0.000,C 90.000,E1 28.537} C_DIS
LIN {X -0.073,Y -215.872,Z 348.141,A 0.000,B 0.000,C 90.000,E1 25.463} C_DIS
LIN {X -0.056,Y -209.882,Z 348.124,A 0.000,B 0.000,C 90.000,E1 22.333} C_DIS
LIN {X 0.039,Y -204.640,Z 348.106,A 0.000,B 0.000,C 90.000,E1 19.141} C_DIS
LIN {X -0.063,Y -200.114,Z 348.089,A 0.000,B 0.000,C 90.000,E1 15.969} C_DIS
LIN {X 0.037,Y -195.352,Z 348.066,A 0.000,B 0.000,C 90.000,E1 11.895} C_DIS
LIN {X 0.017,Y -191.736,Z 348.043,A 0.000,B 0.000,C 90.000,E1 7.814} C_DIS
LIN {X 0.034,Y -188.943,Z 348.016,A 0.000,B 0.000,C 90.000,E1 2.865} C_DIS
LIN {X 0.025,Y -187.990,Z 347.970,A 0.000,B 0.000,C 90.000,E1 354.546} C_DIS
LIN {X -0.039,Y -190.074,Z 347.933,A 0.000,B 0.000,C 90.000,E1 347.937} C_DIS
LIN {X 0.068,Y -193.419,Z 347.905,A 0.000,B 0.000,C 90.000,E1 342.960} C_DIS
LIN {X -0.036,Y -197.388,Z 347.883,A 0.000,B 0.000,C 90.000,E1 338.901} C_DIS
LIN {X -0.023,Y -202.415,Z 347.860,A 0.000,B 0.000,C 90.000,E1 334.845} C_DIS
LIN {X -0.047,Y -208.467,Z 347.838,A 0.000,B 0.000,C 90.000,E1 330.845} C_DIS
LIN {X -0.126,Y -215.443,Z 347.816,A 0.000,B 0.000,C 90.000,E1 326.914} C_DIS
LIN {X -0.062,Y -223.222,Z 347.794,A 0.000,B 0.000,C 90.000,E1 323.004} C_DIS
LIN {X 0.049,Y -229.958,Z 347.777,A 0.000,B 0.000,C 90.000,E1 319.908} C_DIS
LIN {X -0.069,Y -238.589,Z 347.758,A 0.000,B 0.000,C 90.000,E1 316.539} C_DIS
LIN {X 0.068,Y -248.440,Z 347.740,A 0.000,B 0.000,C 90.000,E1 313.176} C_DIS
LIN {X -0.011,Y -259.467,Z 347.722,A 0.000,B 0.000,C 90.000,E1 309.930} C_DIS
LIN {X -0.044,Y -271.290,Z 347.704,A 0.000,B 0.000,C 90.000,E1 306.744} C_DIS
LIN {X -0.055,Y -284.311,Z 347.687,A 0.000,B 0.000,C 90.000,E1 303.627} C_DIS
LIN {X -0.073,Y -293.942,Z 347.675,A 0.000,B 0.000,C 90.000,E1 301.592} C_DIS
LIN {X -0.094,Y -311.530,Z 347.657,A 0.000,B 0.000,C 90.000,E1 298.281} C_DIS
LIN {X 0.165,Y -321.278,Z 347.648,A 0.000,B 0.000,C 90.000,E1 296.616} C_DIS
LIN {X -0.111,Y -340.382,Z 347.632,A 0.000,B 0.000,C 90.000,E1 293.823} C_DIS
LIN {X -0.067,Y -353.822,Z 347.622,A 0.000,B 0.000,C 90.000,E1 291.972} C_DIS
LIN {X -0.070,Y -372.315,Z 347.609,A 0.000,B 0.000,C 90.000,E1 289.577} C_DIS
LIN {X -0.051,Y -394.968,Z 347.594,A 0.000,B 0.000,C 90.000,E1 286.968} C_DIS
LIN {X 0.001,Y -410.313,Z 347.585,A 0.000,B 0.000,C 90.000,E1 285.300} C_DIS
LIN {X -0.187,Y -422.682,Z 347.578,A 0.000,B 0.000,C 90.000,E1 284.008} C_DIS
LIN {X 0.011,Y -430.065,Z 347.573,A 0.000,B 0.000,C 90.000,E1 283.175} C_DIS
LIN {X -0.010,Y -439.215,Z 347.567,A 0.000,B 0.000,C 90.000,E1 282.119} C_DIS
LIN {X -0.111,Y -447.561,Z 347.561,A 0.000,B 0.000,C 90.000,E1 281.074} C_DIS
LIN {X -0.028,Y -455.213,Z 347.556,A 0.000,B 0.000,C 90.000,E1 280.018} C_DIS
LIN {X 0.065,Y -462.315,Z 347.550,A 0.000,B 0.000,C 90.000,E1 278.973} C_DIS
LIN {X 0.018,Y -470.417,Z 347.543,A 0.000,B 0.000,C 90.000,E1 277.701} C_DIS
LIN {X -0.243,Y -476.273,Z 347.537,A 0.000,B 0.000,C 90.000,E1 276.720} C_DIS
LIN {X 0.223,Y -480.153,Z 347.533,A 0.000,B 0.000,C 90.000,E1 275.910} C_DIS
LIN {X -0.100,Y -482.508,Z 347.530,A 0.000,B 0.000,C 90.000,E1 275.448} C_DIS
LIN {X 0.026,Y -484.500,Z 347.527,A 0.000,B 0.000,C 90.000,E1 274.935} C_DIS
LIN {X 0.204,Y -486.096,Z 347.525,A 0.000,B 0.000,C 90.000,E1 274.416} C_DIS
LIN {X -0.095,Y -487.284,Z 347.522,A 0.000,B 0.000,C 90.000,E1 273.955} C_DIS
LIN {X 0.069,Y -488.061,Z 347.519,A 0.000,B 0.000,C 90.000,E1 273.440} C_DIS
LIN {X -0.219,Y -488.488,Z 347.516,A 0.000,B 0.000,C 90.000,E1 272.980} C_DIS
LIN {X -0.040,Y -488.614,Z 347.514,A 0.000,B 0.000,C 90.000,E1 272.465} C_DIS
LIN {X 0.145,Y -488.436,Z 347.511,A 0.000,B 0.000,C 90.000,E1 271.949} C_DIS
LIN {X -0.143,Y -488.039,Z 347.508,A 0.000,B 0.000,C 90.000,E1 271.489} C_DIS
LIN {X 0.042,Y -487.390,Z 347.505,A 0.000,B 0.000,C 90.000,E1 270.974} C_DIS
LIN {X 0.225,Y -486.451,Z 347.503,A 0.000,B 0.000,C 90.000,E1 270.458} C_DIS
LIN {X -0.082,Y -485.086,Z 347.500,A 0.000,B 0.000,C 90.000,E1 270.000} C_DIS
LIN {X 0.091,Y -483.289,Z 347.497,A 0.000,B 0.000,C 90.000,E1 269.484} C_DIS
LIN {X -0.225,Y -480.887,Z 347.494,A 0.000,B 0.000,C 90.000,E1 269.026} C_DIS
LIN {X -0.078,Y -477.731,Z 347.492,A 0.000,B 0.000,C 90.000,E1 268.511} C_DIS
LIN {X 0.065,Y -473.610,Z 347.489,A 0.000,B 0.000,C 90.000,E1 267.993} C_DIS
LIN {X 0.171,Y -468.433,Z 347.486,A 0.000,B 0.000,C 90.000,E1 267.478} C_DIS
LIN {X 0.056,Y -462.170,Z 347.483,A 0.000,B 0.000,C 90.000,E1 267.020} C_DIS
LIN {X -0.136,Y -458.911,Z 347.482,A 0.000,B 0.000,C 90.000,E1 266.846} C_DIS
LIN {X -0.221,Y -451.792,Z 347.480,A 0.000,B 0.000,C 90.000,E1 266.502} C_DIS
LIN {X -0.095,Y -447.803,Z 347.480,A 0.000,B 0.000,C 90.000,E1 266.331} C_DIS
LIN {X -0.171,Y -439.702,Z 347.478,A 0.000,B 0.000,C 90.000,E1 266.102} C_DIS
LIN {X -0.137,Y -431.121,Z 347.477,A 0.000,B 0.000,C 90.000,E1 265.927} C_DIS
LIN {X 0.073,Y -423.793,Z 347.477,A 0.000,B 0.000,C 90.000,E1 265.812} C_DIS
LIN {X -0.191,Y -415.839,Z 347.477,A 0.000,B 0.000,C 90.000,E1 265.812} C_DIS
LIN {X 0.074,Y -180.913,Z 347.477,A 0.000,B 0.000,C 90.000,E1 265.755} C_DIS
LIN {X -0.008,Y -180.833,Z 347.472,A 0.000,B 0.000,C 90.000,E1 264.894} C_DIS
LIN {X 0.071,Y -178.940,Z 347.443,A 0.000,B 0.000,C 90.000,E1 259.803} C_DIS
LIN {X -0.062,Y -175.990,Z 347.415,A 0.000,B 0.000,C 90.000,E1 254.755} C_DIS
LIN {X 0.053,Y -175.491,Z 347.410,A 0.000,B 0.000,C 90.000,E1 253.866} C_DIS
LIN {X -0.053,Y -172.234,Z 347.387,A 0.000,B 0.000,C 90.000,E1 249.625} C_DIS
LIN {X -0.074,Y -171.712,Z 347.382,A 0.000,B 0.000,C 90.000,E1 248.773} C_DIS
LIN {X 0.011,Y -167.307,Z 347.353,A 0.000,B 0.000,C 90.000,E1 243.563} C_DIS
LIN {X 0.017,Y -166.688,Z 347.348,A 0.000,B 0.000,C 90.000,E1 242.692} C_DIS
LIN {X 0.008,Y -162.669,Z 347.324,A 0.000,B 0.000,C 90.000,E1 238.329} C_DIS
LIN {X -0.019,Y -161.358,Z 347.314,A 0.000,B 0.000,C 90.000,E1 236.580} C_DIS
LIN {X 0.015,Y -157.352,Z 347.290,A 0.000,B 0.000,C 90.000,E1 232.145} C_DIS
LIN {X 0.044,Y -155.340,Z 347.275,A 0.000,B 0.000,C 90.000,E1 229.461} C_DIS
LIN {X -0.026,Y -151.688,Z 347.250,A 0.000,B 0.000,C 90.000,E1 225.000} C_DIS
LIN {X 0.022,Y -150.551,Z 347.240,A 0.000,B 0.000,C 90.000,E1 223.176} C_DIS
LIN {X 0.054,Y -147.277,Z 347.215,A 0.000,B 0.000,C 90.000,E1 218.624} C_DIS
LIN {X 0.027,Y -145.306,Z 347.194,A 0.000,B 0.000,C 90.000,E1 214.978} C_DIS
LIN {X 0.019,Y -142.397,Z 347.164,A 0.000,B 0.000,C 90.000,E1 209.461} C_DIS
LIN {X 0.001,Y -141.378,Z 347.148,A 0.000,B 0.000,C 90.000,E1 206.693} C_DIS
LIN {X 0.042,Y -139.349,Z 347.112,A 0.000,B 0.000,C 90.000,E1 200.174} C_DIS
LIN {X -0.017,Y -138.785,Z 347.097,A 0.000,B 0.000,C 90.000,E1 197.402} C_DIS
LIN {X 0.043,Y -138.344,Z 347.055,A 0.000,B 0.000,C 90.000,E1 189.905} C_DIS
LIN {X 0.063,Y -139.388,Z 347.008,A 0.000,B 0.000,C 90.000,E1 181.489} C_DIS
LIN {X -0.024,Y -141.285,Z 346.972,A 0.000,B 0.000,C 90.000,E1 175.008} C_DIS
LIN {X -0.066,Y -142.648,Z 346.957,A 0.000,B 0.000,C 90.000,E1 172.243} C_DIS
LIN {X 0.026,Y -144.986,Z 346.931,A 0.000,B 0.000,C 90.000,E1 167.589} C_DIS
LIN {X 0.016,Y -147.613,Z 346.911,A 0.000,B 0.000,C 90.000,E1 163.921} C_DIS
LIN {X -0.047,Y -150.237,Z 346.890,A 0.000,B 0.000,C 90.000,E1 160.296} C_DIS
LIN {X -0.031,Y -153.630,Z 346.870,A 0.000,B 0.000,C 90.000,E1 156.666} C_DIS
LIN {X 0.027,Y -157.045,Z 346.850,A 0.000,B 0.000,C 90.000,E1 153.050} C_DIS
LIN {X 0.025,Y -161.172,Z 346.831,A 0.000,B 0.000,C 90.000,E1 149.488} C_DIS
LIN {X -0.031,Y -163.267,Z 346.821,A 0.000,B 0.000,C 90.000,E1 147.740} C_DIS
LIN {X 0.067,Y -167.707,Z 346.801,A 0.000,B 0.000,C 90.000,E1 144.196} C_DIS
LIN {X -0.020,Y -171.527,Z 346.787,A 0.000,B 0.000,C 90.000,E1 141.618} C_DIS
LIN {X 0.023,Y -176.466,Z 346.768,A 0.000,B 0.000,C 90.000,E1 138.162} C_DIS
LIN {X -0.107,Y -180.763,Z 346.753,A 0.000,B 0.000,C 90.000,E1 135.648} C_DIS
LIN {X 0.010,Y -186.169,Z 346.735,A 0.000,B 0.000,C 90.000,E1 132.243} C_DIS
LIN {X 0.076,Y -190.806,Z 346.721,A 0.000,B 0.000,C 90.000,E1 129.725} C_DIS
LIN {X -0.006,Y -196.564,Z 346.703,A 0.000,B 0.000,C 90.000,E1 126.457} C_DIS
LIN {X 0.043,Y -200.381,Z 346.692,A 0.000,B 0.000,C 90.000,E1 124.532} C_DIS
LIN {X 0.029,Y -300.925,Z 346.692,A 0.000,B 0.000,C 90.000,E1 124.532} C_DIS
LIN {X 0.051,Y -302.991,Z 346.692,A 0.000,B 0.000,C 90.000,E1 124.485} C_DIS
LIN {X 0.046,Y -307.499,Z 346.690,A 0.000,B 0.000,C 90.000,E1 124.246} C_DIS
LIN {X 0.122,Y -310.086,Z 346.689,A 0.000,B 0.000,C 90.000,E1 123.992} C_DIS
LIN {X -0.086,Y -313.851,Z 346.686,A 0.000,B 0.000,C 90.000,E1 123.499} C_DIS
LIN {X -0.038,Y -315.460,Z 346.684,A 0.000,B 0.000,C 90.000,E1 123.166} C_DIS
LIN {X -0.122,Y -318.951,Z 346.679,A 0.000,B 0.000,C 90.000,E1 122.212} C_DIS
LIN {X -0.041,Y -329.763,Z 346.663,A 0.000,B 0.000,C 90.000,E1 119.333} C_DIS
LIN {X 0.161,Y -341.970,Z 346.647,A 0.000,B 0.000,C 90.000,E1 116.488} C_DIS
LIN {X -0.075,Y -354.080,Z 346.634,A 0.000,B 0.000,C 90.000,E1 114.079} C_DIS
LIN {X 0.032,Y -367.466,Z 346.620,A 0.000,B 0.000,C 90.000,E1 111.663} C_DIS
LIN {X -0.003,Y -382.225,Z 346.607,A 0.000,B 0.000,C 90.000,E1 109.322} C_DIS
LIN {X -0.056,Y -398.468,Z 346.595,A 0.000,B 0.000,C 90.000,E1 107.040} C_DIS
LIN {X 0.190,Y -416.314,Z 346.582,A 0.000,B 0.000,C 90.000,E1 104.773} C_DIS
LIN {X -0.088,Y -435.814,Z 346.570,A 0.000,B 0.000,C 90.000,E1 102.647} C_DIS
LIN {X 0.237,Y -456.127,Z 346.559,A 0.000,B 0.000,C 90.000,E1 100.602} C_DIS
LIN {X 0.085,Y -479.592,Z 346.548,A 0.000,B 0.000,C 90.000,E1 98.568} C_DIS
LIN {X -0.112,Y -492.874,Z 346.542,A 0.000,B 0.000,C 90.000,E1 97.530} C_DIS
LIN {X -0.209,Y -496.659,Z 346.539,A 0.000,B 0.000,C 90.000,E1 97.125} C_DIS
LIN {X 0.190,Y -498.142,Z 346.538,A 0.000,B 0.000,C 90.000,E1 96.834} C_DIS
LIN {X 0.035,Y -499.246,Z 346.537,A 0.000,B 0.000,C 90.000,E1 96.606} C_DIS
LIN {X -0.186,Y -500.532,Z 346.534,A 0.000,B 0.000,C 90.000,E1 96.144} C_DIS
LIN {X 0.096,Y -500.781,Z 346.531,A 0.000,B 0.000,C 90.000,E1 95.625} C_DIS
LIN {X -0.114,Y -500.028,Z 346.529,A 0.000,B 0.000,C 90.000,E1 95.163} C_DIS
LIN {X 0.171,Y -498.143,Z 346.526,A 0.000,B 0.000,C 90.000,E1 94.645} C_DIS
LIN {X -0.081,Y -494.935,Z 346.523,A 0.000,B 0.000,C 90.000,E1 94.188} C_DIS
LIN {X -0.106,Y -487.463,Z 346.518,A 0.000,B 0.000,C 90.000,E1 93.212} C_DIS
LIN {X -0.053,Y -475.386,Z 346.510,A 0.000,B 0.000,C 90.000,E1 91.718} C_DIS
LIN {X 0.071,Y -453.975,Z 346.494,A 0.000,B 0.000,C 90.000,E1 88.912} C_DIS
LIN {X -0.055,Y -439.698,Z 346.482,A 0.000,B 0.000,C 90.000,E1 86.846} C_DIS
LIN {X -0.201,Y -423.297,Z 346.468,A 0.000,B 0.000,C 90.000,E1 84.204} C_DIS
LIN {X 0.139,Y -408.177,Z 346.453,A 0.000,B 0.000,C 90.000,E1 81.432} C_DIS
LIN {X 0.063,Y -396.568,Z 346.440,A 0.000,B 0.000,C 90.000,E1 79.218} C_DIS
LIN {X 0.136,Y -386.376,Z 346.429,A 0.000,B 0.000,C 90.000,E1 77.229} C_DIS
LIN {X 0.072,Y -376.199,Z 346.418,A 0.000,B 0.000,C 90.000,E1 75.227} C_DIS
LIN {X -0.033,Y -364.644,Z 346.405,A 0.000,B 0.000,C 90.000,E1 72.906} C_DIS
LIN {X 0.208,Y -354.388,Z 346.393,A 0.000,B 0.000,C 90.000,E1 70.786} C_DIS
LIN {X -0.058,Y -339.974,Z 346.377,A 0.000,B 0.000,C 90.000,E1 67.794} C_DIS
LIN {X 0.071,Y -326.741,Z 346.359,A 0.000,B 0.000,C 90.000,E1 64.665} C_DIS
LIN {X 0.009,Y -315.961,Z 346.343,A 0.000,B 0.000,C 90.000,E1 61.820} C_DIS
LIN {X 0.008,Y -304.609,Z 346.325,A 0.000,B 0.000,C 90.000,E1 58.584} C_DIS
LIN {X -0.093,Y -293.102,Z 346.305,A 0.000,B 0.000,C 90.000,E1 54.975} C_DIS
LIN {X -0.115,Y -283.392,Z 346.287,A 0.000,B 0.000,C 90.000,E1 51.618} C_DIS
LIN {X 0.044,Y -275.914,Z 346.271,A 0.000,B 0.000,C 90.000,E1 48.852} C_DIS
LIN {X 0.165,Y -268.314,Z 346.256,A 0.000,B 0.000,C 90.000,E1 46.053} C_DIS
LIN {X -0.103,Y -260.796,Z 346.240,A 0.000,B 0.000,C 90.000,E1 43.299} C_DIS
LIN {X -0.039,Y -255.085,Z 346.229,A 0.000,B 0.000,C 90.000,E1 41.148} C_DIS
LIN {X -0.052,Y -249.322,Z 346.217,A 0.000,B 0.000,C 90.000,E1 38.991} C_DIS
LIN {X 0.019,Y -243.410,Z 346.204,A 0.000,B 0.000,C 90.000,E1 36.790} C_DIS
LIN {X 0.029,Y -235.573,Z 346.188,A 0.000,B 0.000,C 90.000,E1 33.833} C_DIS
LIN {X 0.009,Y -226.203,Z 346.167,A 0.000,B 0.000,C 90.000,E1 30.079} C_DIS
LIN {X 0.082,Y -219.293,Z 346.150,A 0.000,B 0.000,C 90.000,E1 27.001} C_DIS
LIN {X 0.074,Y -212.933,Z 346.133,A 0.000,B 0.000,C 90.000,E1 23.898} C_DIS
LIN {X -0.064,Y -207.307,Z 346.115,A 0.000,B 0.000,C 90.000,E1 20.791} C_DIS
LIN {X 0.023,Y -202.407,Z 346.098,A 0.000,B 0.000,C 90.000,E1 17.583} C_DIS
LIN {X -0.094,Y -197.268,Z 346.075,A 0.000,B 0.000,C 90.000,E1 13.592} C_DIS
LIN {X -0.019,Y -193.120,Z 346.053,A 0.000,B 0.000,C 90.000,E1 9.500} C_DIS
LIN {X -0.076,Y -189.789,Z 346.025,A 0.000,B 0.000,C 90.000,E1 4.588} C_DIS
LIN {X 0.076,Y -187.844,Z 345.984,A 0.000,B 0.000,C 90.000,E1 357.020} C_DIS
LIN {X -0.012,Y -189.710,Z 345.938,A 0.000,B 0.000,C 90.000,E1 348.757} C_DIS
LIN {X 0.031,Y -192.777,Z 345.910,A 0.000,B 0.000,C 90.000,E1 343.795} C_DIS
LIN {X 0.031,Y -196.501,Z 345.887,A 0.000,B 0.000,C 90.000,E1 339.699} C_DIS
LIN {X -0.063,Y -201.301,Z 345.865,A 0.000,B 0.000,C 90.000,E1 335.665} C_DIS
LIN {X -0.036,Y -207.163,Z 345.842,A 0.000,B 0.000,C 90.000,E1 331.641} C_DIS
LIN {X -0.002,Y -212.504,Z 345.825,A 0.000,B 0.000,C 90.000,E1 328.456} C_DIS
LIN {X -0.090,Y -219.999,Z 345.803,A 0.000,B 0.000,C 90.000,E1 324.562} C_DIS
LIN {X 0.024,Y -228.121,Z 345.782,A 0.000,B 0.000,C 90.000,E1 320.678} C_DIS
LIN {X 0.019,Y -236.484,Z 345.763,A 0.000,B 0.000,C 90.000,E1 317.268} C_DIS
LIN {X -0.089,Y -246.073,Z 345.744,A 0.000,B 0.000,C 90.000,E1 313.947} C_DIS
LIN {X 0.119,Y -256.927,Z 345.726,A 0.000,B 0.000,C 90.000,E1 310.620} C_DIS
LIN {X -0.026,Y -268.584,Z 345.708,A 0.000,B 0.000,C 90.000,E1 307.443} C_DIS
LIN {X -0.118,Y -281.376,Z 345.691,A 0.000,B 0.000,C 90.000,E1 304.326} C_DIS
LIN {X -0.037,Y -290.724,Z 345.679,A 0.000,B 0.000,C 90.000,E1 302.260} C_DIS
LIN {X -0.159,Y -308.067,Z 345.661,A 0.000,B 0.000,C 90.000,E1 298.949} C_DIS
LIN {X -0.094,Y -317.446,Z 345.652,A 0.000,B 0.000,C 90.000,E1 297.308} C_DIS
LIN {X -0.082,Y -338.474,Z 345.634,A 0.000,B 0.000,C 90.000,E1 294.131} C_DIS
LIN {X -0.077,Y -351.867,Z 345.624,A 0.000,B 0.000,C 90.000,E1 292.280} C_DIS
LIN {X -0.041,Y -372.581,Z 345.609,A 0.000,B 0.000,C 90.000,E1 289.577} C_DIS
LIN {X -0.152,Y -395.258,Z 345.594,A 0.000,B 0.000,C 90.000,E1 286.985} C_DIS
LIN {X -0.045,Y -410.607,Z 345.585,A 0.000,B 0.000,C 90.000,E1 285.300} C_DIS
LIN {X -0.209,Y -420.737,Z 345.579,A 0.000,B 0.000,C 90.000,E1 284.245} C_DIS
LIN {X 0.129,Y -430.589,Z 345.573,A 0.000,B 0.000,C 90.000,E1 283.119} C_DIS
LIN {X 0.039,Y -439.702,Z 345.567,A 0.000,B 0.000,C 90.000,E1 282.063} C_DIS
LIN {X 0.032,Y -447.940,Z 345.561,A 0.000,B 0.000,C 90.000,E1 281.007} C_DIS
LIN {X 0.038,Y -455.541,Z 345.555,A 0.000,B 0.000,C 90.000,E1 279.962} C_DIS
LIN {X 0.136,Y -462.564,Z 345.550,A 0.000,B 0.000,C 90.000,E1 278.916} C_DIS
LIN {X -0.212,Y -469.080,Z 345.544,A 0.000,B 0.000,C 90.000,E1 277.936} C_DIS
LIN {X 0.043,Y -475.044,Z 345.538,A 0.000,B 0.000,C 90.000,E1 276.891} C_DIS
LIN {X -0.026,Y -479.063,Z 345.534,A 0.000,B 0.000,C 90.000,E1 276.144} C_DIS
LIN {X -0.014,Y -482.606,Z 345.530,A 0.000,B 0.000,C 90.000,E1 275.391} C_DIS
LIN {X 0.115,Y -484.551,Z 345.527,A 0.000,B 0.000,C 90.000,E1 274.878} C_DIS
LIN {X -0.191,Y -486.099,Z 345.524,A 0.000,B 0.000,C 90.000,E1 274.416} C_DIS
LIN {X -0.004,Y -487.232,Z 345.522,A 0.000,B 0.000,C 90.000,E1 273.898} C_DIS
LIN {X 0.160,Y -487.950,Z 345.519,A 0.000,B 0.000,C 90.000,E1 273.383} C_DIS
LIN {X -0.128,Y -488.374,Z 345.516,A 0.000,B 0.000,C 90.000,E1 272.922} C_DIS
LIN {X 0.051,Y -488.444,Z 345.513,A 0.000,B 0.000,C 90.000,E1 272.407} C_DIS
LIN {X 0.235,Y -488.257,Z 345.511,A 0.000,B 0.000,C 90.000,E1 271.892} C_DIS
LIN {X -0.054,Y -487.871,Z 345.508,A 0.000,B 0.000,C 90.000,E1 271.432} C_DIS
LIN {X 0.130,Y -487.218,Z 345.505,A 0.000,B 0.000,C 90.000,E1 270.917} C_DIS
LIN {X -0.175,Y -486.272,Z 345.502,A 0.000,B 0.000,C 90.000,E1 270.458} C_DIS
LIN {X 0.004,Y -484.908,Z 345.500,A 0.000,B 0.000,C 90.000,E1 269.943} C_DIS
LIN {X 0.176,Y -483.102,Z 345.497,A 0.000,B 0.000,C 90.000,E1 269.427} C_DIS
LIN {X -0.143,Y -480.597,Z 345.494,A 0.000,B 0.000,C 90.000,E1 268.969} C_DIS
LIN {X 0.169,Y -479.146,Z 345.493,A 0.000,B 0.000,C 90.000,E1 268.682} C_DIS
LIN {X -0.172,Y -475.488,Z 345.490,A 0.000,B 0.000,C 90.000,E1 268.224} C_DIS
LIN {X -0.038,Y -470.744,Z 345.487,A 0.000,B 0.000,C 90.000,E1 267.707} C_DIS
LIN {X -0.220,Y -467.924,Z 345.486,A 0.000,B 0.000,C 90.000,E1 267.478} C_DIS
LIN {X -0.230,Y -465.021,Z 345.485,A 0.000,B 0.000,C 90.000,E1 267.249} C_DIS
LIN {X -0.239,Y -461.747,Z 345.483,A 0.000,B 0.000,C 90.000,E1 267.020} C_DIS
LIN {X 0.055,Y -458.474,Z 345.482,A 0.000,B 0.000,C 90.000,E1 266.788} C_DIS
LIN {X -0.135,Y -454.738,Z 345.481,A 0.000,B 0.000,C 90.000,E1 266.617} C_DIS
LIN {X 0.133,Y -447.203,Z 345.479,A 0.000,B 0.000,C 90.000,E1 266.274} C_DIS
LIN {X 0.086,Y -439.155,Z 345.478,A 0.000,B 0.000,C 90.000,E1 266.045} C_DIS
LIN {X 0.153,Y -430.624,Z 345.477,A 0.000,B 0.000,C 90.000,E1 265.869} C_DIS
LIN {X -0.144,Y -420.774,Z 345.477,A 0.000,B 0.000,C 90.000,E1 265.812} C_DIS
LIN {X 0.212,Y -418.945,Z 345.477,A 0.000,B 0.000,C 90.000,E1 265.755} C_DIS
LIN {X 0.064,Y -180.913,Z 345.477,A 0.000,B 0.000,C 90.000,E1 265.755} C_DIS
LIN {X -0.080,Y -180.788,Z 345.471,A 0.000,B 0.000,C 90.000,E1 264.780} C_DIS
LIN {X 0.020,Y -178.804,Z 345.442,A 0.000,B 0.000,C 90.000,E1 259.511} C_DIS
LIN {X 0.096,Y -175.850,Z 345.413,A 0.000,B 0.000,C 90.000,E1 254.393} C_DIS
LIN {X 0.056,Y -172.585,Z 345.390,A 0.000,B 0.000,C 90.000,E1 250.134} C_DIS
LIN {X 0.072,Y -171.475,Z 345.380,A 0.000,B 0.000,C 90.000,E1 248.411} C_DIS
LIN {X 0.051,Y -167.705,Z 345.356,A 0.000,B 0.000,C 90.000,E1 244.101} C_DIS
LIN {X 0.064,Y -166.392,Z 345.347,A 0.000,B 0.000,C 90.000,E1 242.359} C_DIS
LIN {X 0.055,Y -163.118,Z 345.327,A 0.000,B 0.000,C 90.000,E1 238.869} C_DIS
LIN {X 0.106,Y -161.069,Z 345.313,A 0.000,B 0.000,C 90.000,E1 236.215} C_DIS
LIN {X -0.008,Y -157.802,Z 345.293,A 0.000,B 0.000,C 90.000,E1 232.718} C_DIS
LIN {X -0.070,Y -155.837,Z 345.278,A 0.000,B 0.000,C 90.000,E1 230.070} C_DIS
LIN {X -0.012,Y -152.088,Z 345.253,A 0.000,B 0.000,C 90.000,E1 225.567} C_DIS
LIN {X 0.006,Y -150.337,Z 345.238,A 0.000,B 0.000,C 90.000,E1 222.852} C_DIS
LIN {X 0.027,Y -147.076,Z 345.213,A 0.000,B 0.000,C 90.000,E1 218.302} C_DIS
LIN {X -0.068,Y -145.651,Z 345.198,A 0.000,B 0.000,C 90.000,E1 215.598} C_DIS
LIN {X -0.065,Y -143.033,Z 345.172,A 0.000,B 0.000,C 90.000,E1 211.003} C_DIS
LIN {X 0.062,Y -141.658,Z 345.152,A 0.000,B 0.000,C 90.000,E1 207.257} C_DIS
LIN {X -0.019,Y -139.447,Z 345.115,A 0.000,B 0.000,C 90.000,E1 200.791} C_DIS
LIN {X 0.034,Y -139.181,Z 345.105,A 0.000,B 0.000,C 90.000,E1 198.906} C_DIS
LIN {X 0.062,Y -138.320,Z 345.053,A 0.000,B 0.000,C 90.000,E1 189.557} C_DIS
LIN {X -0.068,Y -139.465,Z 345.007,A 0.000,B 0.000,C 90.000,E1 181.203} C_DIS
LIN {X 0.013,Y -141.029,Z 344.975,A 0.000,B 0.000,C 90.000,E1 175.584} C_DIS
LIN {X -0.033,Y -142.395,Z 344.960,A 0.000,B 0.000,C 90.000,E1 172.818} C_DIS
LIN {X 0.029,Y -144.627,Z 344.934,A 0.000,B 0.000,C 90.000,E1 168.173} C_DIS
LIN {X -0.052,Y -147.822,Z 344.909,A 0.000,B 0.000,C 90.000,E1 163.614} C_DIS
LIN {X 0.034,Y -150.513,Z 344.889,A 0.000,B 0.000,C 90.000,E1 159.934} C_DIS
LIN {X 0.055,Y -153.974,Z 344.868,A 0.000,B 0.000,C 90.000,E1 156.305} C_DIS
LIN {X -0.025,Y -157.386,Z 344.849,A 0.000,B 0.000,C 90.000,E1 152.743} C_DIS
LIN {X -0.082,Y -161.590,Z 344.829,A 0.000,B 0.000,C 90.000,E1 149.203} C_DIS
LIN {X -0.072,Y -165.787,Z 344.809,A 0.000,B 0.000,C 90.000,E1 145.674} C_DIS
LIN {X -0.087,Y -170.748,Z 344.790,A 0.000,B 0.000,C 90.000,E1 142.190} C_DIS
LIN {X 0.072,Y -175.621,Z 344.771,A 0.000,B 0.000,C 90.000,E1 138.690} C_DIS
LIN {X -0.059,Y -181.236,Z 344.752,A 0.000,B 0.000,C 90.000,E1 135.324} C_DIS
LIN {X 0.072,Y -186.706,Z 344.733,A 0.000,B 0.000,C 90.000,E1 131.919} C_DIS
LIN {X 0.024,Y -191.305,Z 344.719,A 0.000,B 0.000,C 90.000,E1 129.439} C_DIS
LIN {X -0.045,Y -197.135,Z 344.701,A 0.000,B 0.000,C 90.000,E1 126.171} C_DIS
LIN {X 0.061,Y -200.464,Z 344.692,A 0.000,B 0.000,C 90.000,E1 124.485} C_DIS
LIN {X 0.038,Y -300.989,Z 344.692,A 0.000,B 0.000,C 90.000,E1 124.485} C_DIS
LIN {X 0.046,Y -302.660,Z 344.691,A 0.000,B 0.000,C 90.000,E1 124.452} C_DIS
LIN {X -0.013,Y -306.680,Z 344.690,A 0.000,B 0.000,C 90.000,E1 124.278} C_DIS
LIN {X -0.154,Y -309.005,Z 344.689,A 0.000,B 0.000,C 90.000,E1 124.119} C_DIS
LIN {X 0.075,Y -312.203,Z 344.687,A 0.000,B 0.000,C 90.000,E1 123.706} C_DIS
LIN {X -0.078,Y -314.156,Z 344.686,A 0.000,B 0.000,C 90.000,E1 123.420} C_DIS
LIN {X 0.030,Y -315.683,Z 344.684,A 0.000,B 0.000,C 90.000,E1 123.086} C_DIS
LIN {X 0.111,Y -321.451,Z 344.675,A 0.000,B 0.000,C 90.000,E1 121.465} C_DIS
LIN {X 0.101,Y -332.596,Z 344.659,A 0.000,B 0.000,C 90.000,E1 118.615} C_DIS
LIN {X -0.066,Y -345.158,Z 344.644,A 0.000,B 0.000,C 90.000,E1 115.848} C_DIS
LIN {X 0.093,Y -357.608,Z 344.630,A 0.000,B 0.000,C 90.000,E1 113.387} C_DIS
LIN {X -0.186,Y -371.362,Z 344.617,A 0.000,B 0.000,C 90.000,E1 111.046} C_DIS
LIN {X 0.104,Y -386.518,Z 344.604,A 0.000,B 0.000,C 90.000,E1 108.671} C_DIS
LIN {X -0.213,Y -403.189,Z 344.591,A 0.000,B 0.000,C 90.000,E1 106.441} C_DIS
LIN {X 0.041,Y -421.498,Z 344.579,A 0.000,B 0.000,C 90.000,E1 104.189} C_DIS
LIN {X 0.038,Y -441.305,Z 344.567,A 0.000,B 0.000,C 90.000,E1 102.063} C_DIS
LIN {X -0.234,Y -461.770,Z 344.556,A 0.000,B 0.000,C 90.000,E1 100.141} C_DIS
LIN {X -0.024,Y -485.411,Z 344.545,A 0.000,B 0.000,C 90.000,E1 98.106} C_DIS
LIN {X 0.026,Y -493.341,Z 344.542,A 0.000,B 0.000,C 90.000,E1 97.473} C_DIS
LIN {X -0.216,Y -495.397,Z 344.540,A 0.000,B 0.000,C 90.000,E1 97.296} C_DIS
LIN {X 0.146,Y -497.227,Z 344.539,A 0.000,B 0.000,C 90.000,E1 97.011} C_DIS
LIN {X 0.079,Y -498.604,Z 344.538,A 0.000,B 0.000,C 90.000,E1 96.777} C_DIS
LIN {X -0.149,Y -500.356,Z 344.535,A 0.000,B 0.000,C 90.000,E1 96.315} C_DIS
LIN {X 0.127,Y -501.000,Z 344.532,A 0.000,B 0.000,C 90.000,E1 95.796} C_DIS
LIN {X -0.085,Y -500.646,Z 344.530,A 0.000,B 0.000,C 90.000,E1 95.334} C_DIS
LIN {X 0.160,Y -499.237,Z 344.527,A 0.000,B 0.000,C 90.000,E1 94.821} C_DIS
LIN {X 0.075,Y -498.061,Z 344.526,A 0.000,B 0.000,C 90.000,E1 94.588} C_DIS
LIN {X -0.180,Y -494.742,Z 344.523,A 0.000,B 0.000,C 90.000,E1 94.131} C_DIS
LIN {X -0.178,Y -487.216,Z 344.517,A 0.000,B 0.000,C 90.000,E1 93.151} C_DIS
LIN {X -0.155,Y -475.123,Z 344.509,A 0.000,B 0.000,C 90.000,E1 91.661} C_DIS
LIN {X -0.028,Y -453.720,Z 344.494,A 0.000,B 0.000,C 90.000,E1 88.854} C_DIS
LIN {X -0.157,Y -439.471,Z 344.482,A 0.000,B 0.000,C 90.000,E1 86.788} C_DIS
LIN {X 0.114,Y -423.086,Z 344.467,A 0.000,B 0.000,C 90.000,E1 84.090} C_DIS
LIN {X 0.027,Y -407.999,Z 344.452,A 0.000,B 0.000,C 90.000,E1 81.376} C_DIS
LIN {X -0.051,Y -396.418,Z 344.440,A 0.000,B 0.000,C 90.000,E1 79.162} C_DIS
LIN {X 0.015,Y -386.223,Z 344.429,A 0.000,B 0.000,C 90.000,E1 77.173} C_DIS
LIN {X -0.050,Y -376.055,Z 344.418,A 0.000,B 0.000,C 90.000,E1 75.172} C_DIS
LIN {X -0.051,Y -364.470,Z 344.405,A 0.000,B 0.000,C 90.000,E1 72.834} C_DIS
LIN {X 0.076,Y -354.223,Z 344.393,A 0.000,B 0.000,C 90.000,E1 70.732} C_DIS
LIN {X -0.068,Y -339.804,Z 344.376,A 0.000,B 0.000,C 90.000,E1 67.720} C_DIS
LIN {X -0.038,Y -327.871,Z 344.361,A 0.000,B 0.000,C 90.000,E1 64.921} C_DIS
LIN {X -0.138,Y -315.868,Z 344.343,A 0.000,B 0.000,C 90.000,E1 61.769} C_DIS
LIN {X -0.145,Y -304.538,Z 344.325,A 0.000,B 0.000,C 90.000,E1 58.535} C_DIS
LIN {X 0.150,Y -294.063,Z 344.307,A 0.000,B 0.000,C 90.000,E1 55.182} C_DIS
LIN {X 0.153,Y -284.298,Z 344.288,A 0.000,B 0.000,C 90.000,E1 51.823} C_DIS
LIN {X -0.059,Y -276.825,Z 344.273,A 0.000,B 0.000,C 90.000,E1 49.138} C_DIS
LIN {X -0.093,Y -269.214,Z 344.258,A 0.000,B 0.000,C 90.000,E1 46.377} C_DIS
LIN {X 0.038,Y -261.680,Z 344.242,A 0.000,B 0.000,C 90.000,E1 43.542} C_DIS
LIN {X -0.075,Y -255.991,Z 344.230,A 0.000,B 0.000,C 90.000,E1 41.434} C_DIS
LIN {X -0.073,Y -250.252,Z 344.218,A 0.000,B 0.000,C 90.000,E1 39.277} C_DIS
LIN {X 0.014,Y -244.339,Z 344.206,A 0.000,B 0.000,C 90.000,E1 37.076} C_DIS
LIN {X 0.048,Y -236.501,Z 344.190,A 0.000,B 0.000,C 90.000,E1 34.119} C_DIS
LIN {X -0.020,Y -227.067,Z 344.169,A 0.000,B 0.000,C 90.000,E1 30.384} C_DIS
LIN {X 0.058,Y -218.409,Z 344.148,A 0.000,B 0.000,C 90.000,E1 26.539} C_DIS
LIN {X -0.062,Y -212.111,Z 344.130,A 0.000,B 0.000,C 90.000,E1 23.462} C_DIS
LIN {X -0.024,Y -206.602,Z 344.113,A 0.000,B 0.000,C 90.000,E1 20.301} C_DIS
LIN {X 0.043,Y -201.819,Z 344.095,A 0.000,B 0.000,C 90.000,E1 17.094} C_DIS
LIN {X 0.043,Y -196.791,Z 344.073,A 0.000,B 0.000,C 90.000,E1 13.063} C_DIS
LIN {X 0.099,Y -192.811,Z 344.050,A 0.000,B 0.000,C 90.000,E1 8.973} C_DIS
LIN {X -0.013,Y -189.646,Z 344.023,A 0.000,B 0.000,C 90.000,E1 4.073} C_DIS
LIN {X 0.030,Y -188.112,Z 343.970,A 0.000,B 0.000,C 90.000,E1 354.546} C_DIS
LIN {X -0.029,Y -190.145,Z 343.933,A 0.000,B 0.000,C 90.000,E1 347.937} C_DIS
LIN {X 0.081,Y -193.473,Z 343.905,A 0.000,B 0.000,C 90.000,E1 342.960} C_DIS
LIN {X -0.021,Y -197.382,Z 343.883,A 0.000,B 0.000,C 90.000,E1 338.901} C_DIS
LIN {X -0.008,Y -202.380,Z 343.860,A 0.000,B 0.000,C 90.000,E1 334.845} C_DIS
LIN {X -0.033,Y -208.393,Z 343.838,A 0.000,B 0.000,C 90.000,E1 330.845} C_DIS
LIN {X 0.033,Y -213.904,Z 343.820,A 0.000,B 0.000,C 90.000,E1 327.661} C_DIS
LIN {X -0.073,Y -221.511,Z 343.799,A 0.000,B 0.000,C 90.000,E1 323.783} C_DIS
LIN {X 0.029,Y -228.045,Z 343.782,A 0.000,B 0.000,C 90.000,E1 320.678} C_DIS
LIN {X 0.022,Y -236.428,Z 343.763,A 0.000,B 0.000,C 90.000,E1 317.268} C_DIS
LIN {X -0.089,Y -246.036,Z 343.744,A 0.000,B 0.000,C 90.000,E1 313.947} C_DIS
LIN {X 0.119,Y -256.904,Z 343.726,A 0.000,B 0.000,C 90.000,E1 310.620} C_DIS
LIN {X -0.027,Y -268.588,Z 343.708,A 0.000,B 0.000,C 90.000,E1 307.443} C_DIS
LIN {X -0.118,Y -281.448,Z 343.691,A 0.000,B 0.000,C 90.000,E1 304.326} C_DIS
LIN {X -0.035,Y -290.845,Z 343.679,A 0.000,B 0.000,C 90.000,E1 302.260} C_DIS
LIN {X -0.033,Y -306.433,Z 343.663,A 0.000,B 0.000,C 90.000,E1 299.255} C_DIS
LIN {X -0.086,Y -317.658,Z 343.652,A 0.000,B 0.000,C 90.000,E1 297.308} C_DIS
LIN {X -0.064,Y -338.765,Z 343.634,A 0.000,B 0.000,C 90.000,E1 294.131} C_DIS
LIN {X -0.053,Y -352.156,Z 343.624,A 0.000,B 0.000,C 90.000,E1 292.280} C_DIS
LIN {X -0.006,Y -372.861,Z 343.609,A 0.000,B 0.000,C 90.000,E1 289.577} C_DIS
LIN {X -0.054,Y -395.428,Z 343.594,A 0.000,B 0.000,C 90.000,E1 286.985} C_DIS
LIN {X -0.196,Y -408.216,Z 343.587,A 0.000,B 0.000,C 90.000,E1 285.607} C_DIS
LIN {X 0.045,Y -423.438,Z 343.577,A 0.000,B 0.000,C 90.000,E1 283.939} C_DIS
LIN {X 0.120,Y -430.741,Z 343.573,A 0.000,B 0.000,C 90.000,E1 283.119} C_DIS
LIN {X -0.181,Y -437.609,Z 343.569,A 0.000,B 0.000,C 90.000,E1 282.355} C_DIS
LIN {X -0.004,Y -444.022,Z 343.564,A 0.000,B 0.000,C 90.000,E1 281.535} C_DIS
LIN {X -0.045,Y -451.851,Z 343.558,A 0.000,B 0.000,C 90.000,E1 280.489} C_DIS
LIN {X 0.012,Y -459.119,Z 343.552,A 0.000,B 0.000,C 90.000,E1 279.443} C_DIS
LIN {X -0.008,Y -467.445,Z 343.545,A 0.000,B 0.000,C 90.000,E1 278.163} C_DIS
LIN {X 0.167,Y -473.522,Z 343.540,A 0.000,B 0.000,C 90.000,E1 277.125} C_DIS
LIN {X -0.055,Y -478.975,Z 343.534,A 0.000,B 0.000,C 90.000,E1 276.144} C_DIS
LIN {X -0.043,Y -482.503,Z 343.530,A 0.000,B 0.000,C 90.000,E1 275.391} C_DIS
LIN {X 0.084,Y -484.425,Z 343.527,A 0.000,B 0.000,C 90.000,E1 274.878} C_DIS
LIN {X -0.222,Y -486.017,Z 343.524,A 0.000,B 0.000,C 90.000,E1 274.416} C_DIS
LIN {X -0.036,Y -487.128,Z 343.522,A 0.000,B 0.000,C 90.000,E1 273.898} C_DIS
LIN {X 0.127,Y -487.844,Z 343.519,A 0.000,B 0.000,C 90.000,E1 273.383} C_DIS
LIN {X -0.161,Y -488.223,Z 343.516,A 0.000,B 0.000,C 90.000,E1 272.922} C_DIS
LIN {X 0.017,Y -488.270,Z 343.513,A 0.000,B 0.000,C 90.000,E1 272.407} C_DIS
LIN {X 0.200,Y -488.114,Z 343.511,A 0.000,B 0.000,C 90.000,E1 271.892} C_DIS
LIN {X -0.089,Y -487.713,Z 343.508,A 0.000,B 0.000,C 90.000,E1 271.432} C_DIS
LIN {X 0.093,Y -487.100,Z 343.505,A 0.000,B 0.000,C 90.000,E1 270.917} C_DIS
LIN {X -0.212,Y -486.167,Z 343.502,A 0.000,B 0.000,C 90.000,E1 270.458} C_DIS
LIN {X -0.034,Y -484.889,Z 343.500,A 0.000,B 0.000,C 90.000,E1 269.943} C_DIS
LIN {X 0.138,Y -483.105,Z 343.497,A 0.000,B 0.000,C 90.000,E1 269.427} C_DIS
LIN {X -0.181,Y -480.655,Z 343.494,A 0.000,B 0.000,C 90.000,E1 268.969} C_DIS
LIN {X -0.036,Y -477.474,Z 343.491,A 0.000,B 0.000,C 90.000,E1 268.453} C_DIS
LIN {X 0.107,Y -473.352,Z 343.489,A 0.000,B 0.000,C 90.000,E1 267.936} C_DIS
LIN {X -0.076,Y -470.824,Z 343.487,A 0.000,B 0.000,C 90.000,E1 267.707} C_DIS
LIN {X 0.206,Y -465.159,Z 343.485,A 0.000,B 0.000,C 90.000,E1 267.192} C_DIS
LIN {X 0.202,Y -461.856,Z 343.483,A 0.000,B 0.000,C 90.000,E1 266.963} C_DIS
LIN {X 0.050,Y -458.683,Z 343.482,A 0.000,B 0.000,C 90.000,E1 266.788} C_DIS
LIN {X -0.124,Y -454.917,Z 343.481,A 0.000,B 0.000,C 90.000,E1 266.617} C_DIS
LIN {X 0.182,Y -447.557,Z 343.479,A 0.000,B 0.000,C 90.000,E1 266.274} C_DIS
LIN {X 0.109,Y -439.720,Z 343.478,A 0.000,B 0.000,C 90.000,E1 266.045} C_DIS
LIN {X 0.112,Y -430.849,Z 343.477,A 0.000,B 0.000,C 90.000,E1 265.869} C_DIS
LIN {X -0.106,Y -422.993,Z 343.477,A 0.000,B 0.000,C 90.000,E1 265.812} C_DIS
LIN {X 0.102,Y -415.028,Z 343.477,A 0.000,B 0.000,C 90.000,E1 265.755} C_DIS
LIN {X 0.026,Y -180.912,Z 343.476,A 0.000,B 0.000,C 90.000,E1 265.755} C_DIS
LIN {X -0.047,Y -180.830,Z 343.472,A 0.000,B 0.000,C 90.000,E1 264.894} C_DIS
LIN {X 0.033,Y -178.936,Z 343.443,A 0.000,B 0.000,C 90.000,E1 259.803} C_DIS
LIN {X -0.100,Y -175.985,Z 343.415,A 0.000,B 0.000,C 90.000,E1 254.755} C_DIS
LIN {X 0.015,Y -175.480,Z 343.410,A 0.000,B 0.000,C 90.000,E1 253.866} C_DIS
LIN {X 0.072,Y -172.227,Z 343.387,A 0.000,B 0.000,C 90.000,E1 249.571} C_DIS
LIN {X 0.049,Y -171.703,Z 343.382,A 0.000,B 0.000,C 90.000,E1 248.720} C_DIS
LIN {X -0.025,Y -167.298,Z 343.353,A 0.000,B 0.000,C 90.000,E1 243.563} C_DIS
LIN {X -0.020,Y -166.676,Z 343.348,A 0.000,B 0.000,C 90.000,E1 242.692} C_DIS
LIN {X -0.028,Y -162.659,Z 343.324,A 0.000,B 0.000,C 90.000,E1 238.329} C_DIS
LIN {X 0.034,Y -161.348,Z 343.314,A 0.000,B 0.000,C 90.000,E1 236.548} C_DIS
LIN {X 0.077,Y -157.342,Z 343.290,A 0.000,B 0.000,C 90.000,E1 232.110} C_DIS
LIN {X 0.009,Y -155.328,Z 343.275,A 0.000,B 0.000,C 90.000,E1 229.461} C_DIS
LIN {X -0.061,Y -151.679,Z 343.250,A 0.000,B 0.000,C 90.000,E1 225.000} C_DIS
LIN {X -0.012,Y -150.543,Z 343.240,A 0.000,B 0.000,C 90.000,E1 223.176} C_DIS
LIN {X 0.020,Y -147.269,Z 343.215,A 0.000,B 0.000,C 90.000,E1 218.624} C_DIS
LIN {X -0.007,Y -145.296,Z 343.194,A 0.000,B 0.000,C 90.000,E1 214.978} C_DIS
LIN {X -0.014,Y -142.392,Z 343.164,A 0.000,B 0.000,C 90.000,E1 209.461} C_DIS
LIN {X 0.032,Y -141.373,Z 343.148,A 0.000,B 0.000,C 90.000,E1 206.668} C_DIS
LIN {X 0.009,Y -139.346,Z 343.112,A 0.000,B 0.000,C 90.000,E1 200.174} C_DIS
LIN {X 0.014,Y -139.018,Z 343.102,A 0.000,B 0.000,C 90.000,E1 198.308} C_DIS
LIN {X 0.010,Y -138.343,Z 343.055,A 0.000,B 0.000,C 90.000,E1 189.905} C_DIS
LIN {X 0.030,Y -139.392,Z 343.008,A 0.000,B 0.000,C 90.000,E1 181.489} C_DIS
LIN {X -0.056,Y -141.291,Z 342.972,A 0.000,B 0.000,C 90.000,E1 175.008} C_DIS
LIN {X 0.042,Y -142.654,Z 342.957,A 0.000,B 0.000,C 90.000,E1 172.186} C_DIS
LIN {X -0.008,Y -144.994,Z 342.931,A 0.000,B 0.000,C 90.000,E1 167.589} C_DIS
LIN {X -0.019,Y -147.621,Z 342.911,A 0.000,B 0.000,C 90.000,E1 163.921} C_DIS
LIN {X 0.060,Y -150.248,Z 342.890,A 0.000,B 0.000,C 90.000,E1 160.242} C_DIS
LIN {X -0.067,Y -153.643,Z 342.870,A 0.000,B 0.000,C 90.000,E1 156.666} C_DIS
LIN {X -0.008,Y -157.058,Z 342.850,A 0.000,B 0.000,C 90.000,E1 153.050} C_DIS
LIN {X 0.072,Y -161.188,Z 342.830,A 0.000,B 0.000,C 90.000,E1 149.459} C_DIS
LIN {X 0.020,Y -163.281,Z 342.821,A 0.000,B 0.000,C 90.000,E1 147.709} C_DIS
LIN {X 0.030,Y -167.725,Z 342.801,A 0.000,B 0.000,C 90.000,E1 144.196} C_DIS
LIN {X -0.058,Y -171.543,Z 342.787,A 0.000,B 0.000,C 90.000,E1 141.618} C_DIS
LIN {X -0.015,Y -176.485,Z 342.768,A 0.000,B 0.000,C 90.000,E1 138.162} C_DIS
LIN {X 0.110,Y -180.783,Z 342.753,A 0.000,B 0.000,C 90.000,E1 135.567} C_DIS
LIN {X -0.029,Y -186.190,Z 342.735,A 0.000,B 0.000,C 90.000,E1 132.243} C_DIS
LIN {X 0.035,Y -190.827,Z 342.721,A 0.000,B 0.000,C 90.000,E1 129.725} C_DIS
LIN {X -0.047,Y -196.586,Z 342.702,A 0.000,B 0.000,C 90.000,E1 126.457} C_DIS
LIN {X 0.009,Y -200.558,Z 342.691,A 0.000,B 0.000,C 90.000,E1 124.452} C_DIS
LIN {X -0.033,Y -300.614,Z 342.691,A 0.000,B 0.000,C 90.000,E1 124.452} C_DIS
LIN {X 0.081,Y -302.416,Z 342.691,A 0.000,B 0.000,C 90.000,E1 124.405} C_DIS
LIN {X 0.070,Y -307.037,Z 342.690,A 0.000,B 0.000,C 90.000,E1 124.199} C_DIS
LIN {X 0.058,Y -309.546,Z 342.689,A 0.000,B 0.000,C 90.000,E1 123.992} C_DIS
LIN {X 0.095,Y -313.368,Z 342.686,A 0.000,B 0.000,C 90.000,E1 123.499} C_DIS
LIN {X 0.143,Y -315.149,Z 342.684,A 0.000,B 0.000,C 90.000,E1 123.166} C_DIS
LIN {X -0.075,Y -316.545,Z 342.683,A 0.000,B 0.000,C 90.000,E1 122.880} C_DIS
LIN {X 0.033,Y -328.327,Z 342.665,A 0.000,B 0.000,C 90.000,E1 119.667} C_DIS
LIN {X -0.101,Y -340.355,Z 342.649,A 0.000,B 0.000,C 90.000,E1 116.873} C_DIS
LIN {X 0.082,Y -352.296,Z 342.636,A 0.000,B 0.000,C 90.000,E1 114.387} C_DIS
LIN {X -0.193,Y -365.499,Z 342.622,A 0.000,B 0.000,C 90.000,E1 112.025} C_DIS
LIN {X 0.068,Y -380.063,Z 342.609,A 0.000,B 0.000,C 90.000,E1 109.631} C_DIS
LIN {X 0.086,Y -396.094,Z 342.596,A 0.000,B 0.000,C 90.000,E1 107.330} C_DIS
LIN {X -0.237,Y -413.712,Z 342.584,A 0.000,B 0.000,C 90.000,E1 105.134} C_DIS
LIN {X -0.106,Y -433.010,Z 342.572,A 0.000,B 0.000,C 90.000,E1 102.939} C_DIS
LIN {X 0.021,Y -453.245,Z 342.561,A 0.000,B 0.000,C 90.000,E1 100.894} C_DIS
LIN {X 0.074,Y -474.016,Z 342.550,A 0.000,B 0.000,C 90.000,E1 99.029} C_DIS
LIN {X 0.051,Y -492.594,Z 342.542,A 0.000,B 0.000,C 90.000,E1 97.530} C_DIS
LIN {X 0.020,Y -496.609,Z 342.540,A 0.000,B 0.000,C 90.000,E1 97.125} C_DIS
LIN {X -0.068,Y -498.200,Z 342.538,A 0.000,B 0.000,C 90.000,E1 96.891} C_DIS
LIN {X -0.217,Y -499.391,Z 342.537,A 0.000,B 0.000,C 90.000,E1 96.663} C_DIS
LIN {X 0.058,Y -500.825,Z 342.534,A 0.000,B 0.000,C 90.000,E1 96.144} C_DIS
LIN {X -0.157,Y -501.202,Z 342.531,A 0.000,B 0.000,C 90.000,E1 95.682} C_DIS
LIN {X 0.132,Y -500.581,Z 342.529,A 0.000,B 0.000,C 90.000,E1 95.163} C_DIS
LIN {X -0.077,Y -498.856,Z 342.526,A 0.000,B 0.000,C 90.000,E1 94.702} C_DIS
LIN {X -0.202,Y -497.478,Z 342.525,A 0.000,B 0.000,C 90.000,E1 94.473} C_DIS
LIN {X -0.061,Y -492.142,Z 342.521,A 0.000,B 0.000,C 90.000,E1 93.726} C_DIS
LIN {X -0.119,Y -484.369,Z 342.515,A 0.000,B 0.000,C 90.000,E1 92.751} C_DIS
LIN {X 0.229,Y -466.223,Z 342.503,A 0.000,B 0.000,C 90.000,E1 90.458} C_DIS
LIN {X 0.086,Y -445.600,Z 342.487,A 0.000,B 0.000,C 90.000,E1 87.650} C_DIS
LIN {X -0.196,Y -427.130,Z 342.471,A 0.000,B 0.000,C 90.000,E1 84.780} C_DIS
LIN {X 0.037,Y -408.822,Z 342.453,A 0.000,B 0.000,C 90.000,E1 81.489} C_DIS
LIN {X -0.010,Y -395.808,Z 342.439,A 0.000,B 0.000,C 90.000,E1 78.993} C_DIS
LIN {X 0.120,Y -385.599,Z 342.428,A 0.000,B 0.000,C 90.000,E1 76.992} C_DIS
LIN {X 0.049,Y -373.990,Z 342.415,A 0.000,B 0.000,C 90.000,E1 74.700} C_DIS
LIN {X -0.081,Y -363.820,Z 342.404,A 0.000,B 0.000,C 90.000,E1 72.670} C_DIS
LIN {X 0.137,Y -353.607,Z 342.392,A 0.000,B 0.000,C 90.000,E1 70.550} C_DIS
LIN {X -0.030,Y -339.173,Z 342.375,A 0.000,B 0.000,C 90.000,E1 67.539} C_DIS
LIN {X 0.118,Y -327.346,Z 342.360,A 0.000,B 0.000,C 90.000,E1 64.717} C_DIS
LIN {X -0.072,Y -316.588,Z 342.344,A 0.000,B 0.000,C 90.000,E1 61.897} C_DIS
LIN {X -0.057,Y -305.223,Z 342.326,A 0.000,B 0.000,C 90.000,E1 58.663} C_DIS
LIN {X 0.028,Y -293.697,Z 342.306,A 0.000,B 0.000,C 90.000,E1 55.022} C_DIS
LIN {X 0.030,Y -283.968,Z 342.287,A 0.000,B 0.000,C 90.000,E1 51.662} C_DIS
LIN {X 0.026,Y -276.483,Z 342.272,A 0.000,B 0.000,C 90.000,E1 48.933} C_DIS
LIN {X 0.007,Y -270.746,Z 342.260,A 0.000,B 0.000,C 90.000,E1 46.863} C_DIS
LIN {X 0.172,Y -263.197,Z 342.245,A 0.000,B 0.000,C 90.000,E1 44.028} C_DIS
LIN {X 0.088,Y -257.551,Z 342.233,A 0.000,B 0.000,C 90.000,E1 41.919} C_DIS
LIN {X -0.074,Y -251.805,Z 342.221,A 0.000,B 0.000,C 90.000,E1 39.806} C_DIS
LIN {X 0.047,Y -245.948,Z 342.209,A 0.000,B 0.000,C 90.000,E1 37.604} C_DIS
LIN {X -0.067,Y -238.080,Z 342.193,A 0.000,B 0.000,C 90.000,E1 34.692} C_DIS
LIN {X 0.073,Y -230.412,Z 342.176,A 0.000,B 0.000,C 90.000,E1 31.671} C_DIS
LIN {X -0.024,Y -221.461,Z 342.155,A 0.000,B 0.000,C 90.000,E1 27.897} C_DIS
LIN {X 0.114,Y -214.866,Z 342.138,A 0.000,B 0.000,C 90.000,E1 24.771} C_DIS
LIN {X 0.020,Y -208.982,Z 342.120,A 0.000,B 0.000,C 90.000,E1 21.663} C_DIS
LIN {X 0.027,Y -203.915,Z 342.103,A 0.000,B 0.000,C 90.000,E1 18.489} C_DIS
LIN {X 0.010,Y -198.494,Z 342.080,A 0.000,B 0.000,C 90.000,E1 14.481} C_DIS
LIN {X -0.027,Y -194.167,Z 342.058,A 0.000,B 0.000,C 90.000,E1 10.433} C_DIS
LIN {X 0.046,Y -190.996,Z 342.035,A 0.000,B 0.000,C 90.000,E1 6.315} C_DIS
LIN {X -0.073,Y -188.485,Z 342.003,A 0.000,B 0.000,C 90.000,E1 0.573} C_DIS
LIN {X 0.000,Y -189.784,Z 341.938,A 0.000,B 0.000,C 90.000,E1 348.757} C_DIS
LIN {X 0.045,Y -192.840,Z 341.910,A 0.000,B 0.000,C 90.000,E1 343.795} C_DIS
LIN {X 0.047,Y -196.526,Z 341.887,A 0.000,B 0.000,C 90.000,E1 339.699} C_DIS
LIN {X -0.046,Y -201.286,Z 341.865,A 0.000,B 0.000,C 90.000,E1 335.665} C_DIS
LIN {X -0.019,Y -207.107,Z 341.842,A 0.000,B 0.000,C 90.000,E1 331.641} C_DIS
LIN {X 0.014,Y -212.431,Z 341.825,A 0.000,B 0.000,C 90.000,E1 328.456} C_DIS
LIN {X -0.076,Y -219.888,Z 341.803,A 0.000,B 0.000,C 90.000,E1 324.562} C_DIS
LIN {X 0.035,Y -227.970,Z 341.782,A 0.000,B 0.000,C 90.000,E1 320.678} C_DIS
LIN {X -0.148,Y -236.370,Z 341.763,A 0.000,B 0.000,C 90.000,E1 317.310} C_DIS
LIN {X -0.085,Y -246.000,Z 341.744,A 0.000,B 0.000,C 90.000,E1 313.947} C_DIS
LIN {X 0.122,Y -256.902,Z 341.726,A 0.000,B 0.000,C 90.000,E1 310.620} C_DIS
LIN {X -0.024,Y -268.597,Z 341.708,A 0.000,B 0.000,C 90.000,E1 307.443} C_DIS
LIN {X -0.114,Y -281.529,Z 341.691,A 0.000,B 0.000,C 90.000,E1 304.326} C_DIS
LIN {X -0.051,Y -292.651,Z 341.677,A 0.000,B 0.000,C 90.000,E1 301.926} C_DIS
LIN {X -0.143,Y -308.422,Z 341.661,A 0.000,B 0.000,C 90.000,E1 298.949} C_DIS
LIN {X -0.071,Y -317.871,Z 341.652,A 0.000,B 0.000,C 90.000,E1 297.308} C_DIS
LIN {X -0.042,Y -339.054,Z 341.634,A 0.000,B 0.000,C 90.000,E1 294.131} C_DIS
LIN {X -0.023,Y -352.439,Z 341.624,A 0.000,B 0.000,C 90.000,E1 292.280} C_DIS
LIN {X 0.033,Y -373.150,Z 341.609,A 0.000,B 0.000,C 90.000,E1 289.577} C_DIS
LIN {X 0.051,Y -395.601,Z 341.594,A 0.000,B 0.000,C 90.000,E1 286.985} C_DIS
LIN {X -0.079,Y -408.325,Z 341.587,A 0.000,B 0.000,C 90.000,E1 285.607} C_DIS
LIN {X 0.061,Y -423.467,Z 341.578,A 0.000,B 0.000,C 90.000,E1 283.953} C_DIS
LIN {X -0.187,Y -430.746,Z 341.573,A 0.000,B 0.000,C 90.000,E1 283.175} C_DIS
LIN {X -0.067,Y -437.602,Z 341.569,A 0.000,B 0.000,C 90.000,E1 282.355} C_DIS
LIN {X -0.100,Y -445.933,Z 341.563,A 0.000,B 0.000,C 90.000,E1 281.299} C_DIS
LIN {X -0.121,Y -453.601,Z 341.557,A 0.000,B 0.000,C 90.000,E1 280.254} C_DIS
LIN {X -0.048,Y -460.711,Z 341.551,A 0.000,B 0.000,C 90.000,E1 279.208} C_DIS
LIN {X -0.121,Y -468.871,Z 341.544,A 0.000,B 0.000,C 90.000,E1 277.936} C_DIS
LIN {X 0.132,Y -474.795,Z 341.538,A 0.000,B 0.000,C 90.000,E1 276.891} C_DIS
LIN {X 0.062,Y -478.801,Z 341.534,A 0.000,B 0.000,C 90.000,E1 276.144} C_DIS
LIN {X 0.073,Y -482.338,Z 341.530,A 0.000,B 0.000,C 90.000,E1 275.391} C_DIS
LIN {X 0.200,Y -484.263,Z 341.527,A 0.000,B 0.000,C 90.000,E1 274.878} C_DIS
LIN {X -0.107,Y -485.822,Z 341.524,A 0.000,B 0.000,C 90.000,E1 274.416} C_DIS
LIN {X 0.079,Y -486.956,Z 341.522,A 0.000,B 0.000,C 90.000,E1 273.898} C_DIS
LIN {X -0.246,Y -487.697,Z 341.519,A 0.000,B 0.000,C 90.000,E1 273.440} C_DIS
LIN {X -0.047,Y -488.054,Z 341.516,A 0.000,B 0.000,C 90.000,E1 272.922} C_DIS
LIN {X 0.129,Y -488.134,Z 341.513,A 0.000,B 0.000,C 90.000,E1 272.407} C_DIS
LIN {X -0.176,Y -487.942,Z 341.511,A 0.000,B 0.000,C 90.000,E1 271.949} C_DIS
LIN {X 0.203,Y -487.007,Z 341.505,A 0.000,B 0.000,C 90.000,E1 270.917} C_DIS
LIN {X -0.104,Y -486.144,Z 341.502,A 0.000,B 0.000,C 90.000,E1 270.458} C_DIS
LIN {X 0.074,Y -484.912,Z 341.500,A 0.000,B 0.000,C 90.000,E1 269.943} C_DIS
LIN {X -0.238,Y -483.137,Z 341.497,A 0.000,B 0.000,C 90.000,E1 269.484} C_DIS
LIN {X 0.085,Y -482.074,Z 341.496,A 0.000,B 0.000,C 90.000,E1 269.198} C_DIS
LIN {X -0.240,Y -479.331,Z 341.493,A 0.000,B 0.000,C 90.000,E1 268.740} C_DIS
LIN {X 0.072,Y -477.677,Z 341.491,A 0.000,B 0.000,C 90.000,E1 268.453} C_DIS
LIN {X 0.213,Y -473.593,Z 341.489,A 0.000,B 0.000,C 90.000,E1 267.936} C_DIS
LIN {X -0.151,Y -468.295,Z 341.486,A 0.000,B 0.000,C 90.000,E1 267.478} C_DIS
LIN {X -0.178,Y -465.453,Z 341.485,A 0.000,B 0.000,C 90.000,E1 267.249} C_DIS
LIN {X 0.110,Y -458.962,Z 341.482,A 0.000,B 0.000,C 90.000,E1 266.788} C_DIS
LIN {X 0.092,Y -451.849,Z 341.480,A 0.000,B 0.000,C 90.000,E1 266.445} C_DIS
LIN {X 0.185,Y -444.403,Z 341.479,A 0.000,B 0.000,C 90.000,E1 266.159} C_DIS
LIN {X -0.114,Y -436.289,Z 341.478,A 0.000,B 0.000,C 90.000,E1 265.988} C_DIS
LIN {X 0.098,Y -427.068,Z 341.477,A 0.000,B 0.000,C 90.000,E1 265.812} C_DIS
LIN {X 0.087,Y -419.170,Z 341.476,A 0.000,B 0.000,C 90.000,E1 265.755} C_DIS
LIN {X 0.014,Y -180.912,Z 341.476,A 0.000,B 0.000,C 90.000,E1 265.755} C_DIS
LIN {X 0.084,Y -180.825,Z 341.471,A 0.000,B 0.000,C 90.000,E1 264.837} C_DIS
LIN {X -0.017,Y -178.930,Z 341.443,A 0.000,B 0.000,C 90.000,E1 259.803} C_DIS
LIN {X 0.021,Y -175.978,Z 341.415,A 0.000,B 0.000,C 90.000,E1 254.700} C_DIS
LIN {X -0.034,Y -175.468,Z 341.410,A 0.000,B 0.000,C 90.000,E1 253.866} C_DIS
LIN {X 0.023,Y -172.217,Z 341.387,A 0.000,B 0.000,C 90.000,E1 249.571} C_DIS
LIN {X 0.001,Y -171.693,Z 341.382,A 0.000,B 0.000,C 90.000,E1 248.720} C_DIS
LIN {X 0.077,Y -167.286,Z 341.353,A 0.000,B 0.000,C 90.000,E1 243.512} C_DIS
LIN {X 0.010,Y -166.662,Z 341.348,A 0.000,B 0.000,C 90.000,E1 242.666} C_DIS
LIN {X -0.075,Y -162.645,Z 341.324,A 0.000,B 0.000,C 90.000,E1 238.329} C_DIS
LIN {X -0.012,Y -161.335,Z 341.314,A 0.000,B 0.000,C 90.000,E1 236.548} C_DIS
LIN {X 0.031,Y -157.329,Z 341.290,A 0.000,B 0.000,C 90.000,E1 232.110} C_DIS
LIN {X -0.036,Y -155.311,Z 341.275,A 0.000,B 0.000,C 90.000,E1 229.461} C_DIS
LIN {X 0.002,Y -151.668,Z 341.250,A 0.000,B 0.000,C 90.000,E1 224.960} C_DIS
LIN {X 0.046,Y -150.534,Z 341.240,A 0.000,B 0.000,C 90.000,E1 223.137} C_DIS
LIN {X -0.023,Y -147.259,Z 341.215,A 0.000,B 0.000,C 90.000,E1 218.624} C_DIS
LIN {X 0.033,Y -145.285,Z 341.194,A 0.000,B 0.000,C 90.000,E1 214.945} C_DIS
LIN {X 0.066,Y -142.386,Z 341.164,A 0.000,B 0.000,C 90.000,E1 209.411} C_DIS
LIN {X -0.011,Y -141.364,Z 341.148,A 0.000,B 0.000,C 90.000,E1 206.668} C_DIS
LIN {X -0.033,Y -139.343,Z 341.112,A 0.000,B 0.000,C 90.000,E1 200.174} C_DIS
LIN {X -0.027,Y -139.014,Z 341.102,A 0.000,B 0.000,C 90.000,E1 198.308} C_DIS
LIN {X -0.032,Y -138.342,Z 341.055,A 0.000,B 0.000,C 90.000,E1 189.905} C_DIS
LIN {X -0.012,Y -139.397,Z 341.008,A 0.000,B 0.000,C 90.000,E1 181.489} C_DIS
LIN {X 0.041,Y -141.299,Z 340.972,A 0.000,B 0.000,C 90.000,E1 174.951} C_DIS
LIN {X -0.001,Y -142.661,Z 340.957,A 0.000,B 0.000,C 90.000,E1 172.186} C_DIS
LIN {X -0.051,Y -145.005,Z 340.931,A 0.000,B 0.000,C 90.000,E1 167.589} C_DIS
LIN {X -0.063,Y -147.632,Z 340.911,A 0.000,B 0.000,C 90.000,E1 163.921} C_DIS
LIN {X 0.015,Y -150.262,Z 340.890,A 0.000,B 0.000,C 90.000,E1 160.242} C_DIS
LIN {X 0.030,Y -153.661,Z 340.870,A 0.000,B 0.000,C 90.000,E1 156.613} C_DIS
LIN {X 0.086,Y -157.076,Z 340.850,A 0.000,B 0.000,C 90.000,E1 152.999} C_DIS
LIN {X 0.025,Y -161.209,Z 340.830,A 0.000,B 0.000,C 90.000,E1 149.459} C_DIS
LIN {X -0.028,Y -163.300,Z 340.821,A 0.000,B 0.000,C 90.000,E1 147.709} C_DIS
LIN {X -0.018,Y -167.747,Z 340.801,A 0.000,B 0.000,C 90.000,E1 144.196} C_DIS
LIN {X -0.105,Y -171.564,Z 340.787,A 0.000,B 0.000,C 90.000,E1 141.618} C_DIS
LIN {X -0.065,Y -176.511,Z 340.767,A 0.000,B 0.000,C 90.000,E1 138.162} C_DIS
LIN {X 0.060,Y -180.809,Z 340.753,A 0.000,B 0.000,C 90.000,E1 135.567} C_DIS
LIN {X 0.046,Y -186.217,Z 340.735,A 0.000,B 0.000,C 90.000,E1 132.204} C_DIS
LIN {X -0.016,Y -190.854,Z 340.721,A 0.000,B 0.000,C 90.000,E1 129.725} C_DIS
LIN {X 0.018,Y -196.616,Z 340.702,A 0.000,B 0.000,C 90.000,E1 126.423} C_DIS
LIN {X -0.024,Y -200.666,Z 340.691,A 0.000,B 0.000,C 90.000,E1 124.405} C_DIS
LIN {X -0.072,Y -301.330,Z 340.691,A 0.000,B 0.000,C 90.000,E1 124.405} C_DIS
LIN {X 0.137,Y -303.300,Z 340.691,A 0.000,B 0.000,C 90.000,E1 124.326} C_DIS
LIN {X -0.155,Y -307.071,Z 340.690,A 0.000,B 0.000,C 90.000,E1 124.199} C_DIS
LIN {X -0.023,Y -309.333,Z 340.689,A 0.000,B 0.000,C 90.000,E1 123.992} C_DIS
LIN {X 0.088,Y -313.208,Z 340.686,A 0.000,B 0.000,C 90.000,E1 123.499} C_DIS
LIN {X 0.137,Y -315.058,Z 340.684,A 0.000,B 0.000,C 90.000,E1 123.166} C_DIS
LIN {X -0.079,Y -316.504,Z 340.683,A 0.000,B 0.000,C 90.000,E1 122.880} C_DIS
LIN {X 0.027,Y -328.309,Z 340.665,A 0.000,B 0.000,C 90.000,E1 119.667} C_DIS
LIN {X -0.108,Y -340.338,Z 340.649,A 0.000,B 0.000,C 90.000,E1 116.873} C_DIS
LIN {X 0.074,Y -352.278,Z 340.636,A 0.000,B 0.000,C 90.000,E1 114.387} C_DIS
LIN {X 0.138,Y -365.482,Z 340.622,A 0.000,B 0.000,C 90.000,E1 111.972} C_DIS
LIN {X 0.059,Y -380.047,Z 340.609,A 0.000,B 0.000,C 90.000,E1 109.631} C_DIS
LIN {X 0.076,Y -396.079,Z 340.596,A 0.000,B 0.000,C 90.000,E1 107.330} C_DIS
LIN {X -0.248,Y -413.697,Z 340.584,A 0.000,B 0.000,C 90.000,E1 105.134} C_DIS
LIN {X -0.117,Y -432.996,Z 340.572,A 0.000,B 0.000,C 90.000,E1 102.939} C_DIS
